Yaskawa INFORM job: sSwarf1_multiple_spiral.JBI

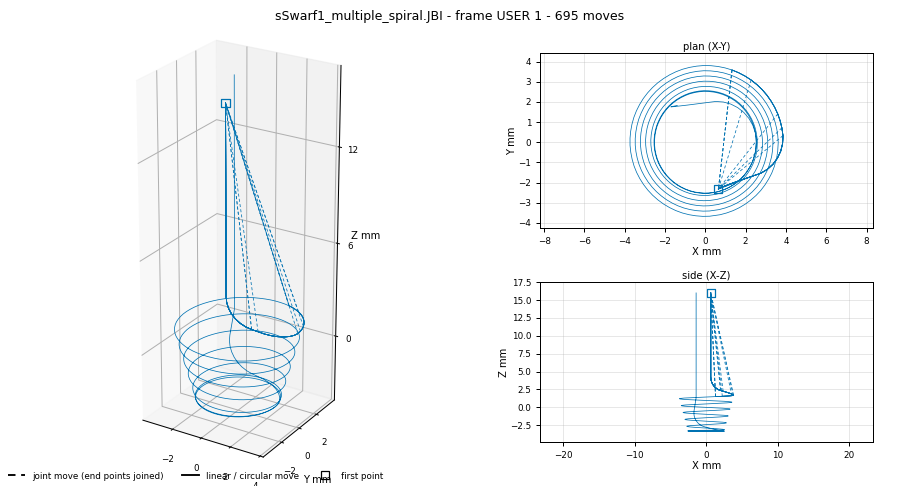
[picture p0: tool path of sSwarf1_multiple_spiral.JBI in frame USER 1, 695 of 695 moves have a stored position in this frame; points joined in program order, loops and branches not executed]
/JOB
//NAME sSwarf1_multiple_spiral
//POS
///NPOS 499,0,0,0,0,0
///USER 1
///TOOL 8
///POSTYPE USER
///RECTAN
///RCONF 1,0,0,0,0,0
C00000=50.999,-29.823,15.536,-90.000,-150.794,-116.565
C00001=50.999,-21.274,0.729,-90.000,-150.794,-116.565
C00002=50.999,-20.274,-1.003,-90.000,-150.794,-116.565
C00003=47.666,-20.274,-1.003,-90.000,-150.794,-116.565
C00004=44.332,-20.274,-1.003,-90.000,-150.794,-116.565
C00005=40.999,-20.274,-1.003,-90.000,-150.794,-116.565
C00006=36.223,-20.274,-1.003,-90.000,-150.794,-116.565
C00007=31.447,-20.274,-1.003,-90.000,-150.794,-116.565
C00008=26.671,-20.274,-1.003,-90.000,-150.794,-116.565
C00009=21.896,-20.274,-1.003,-90.000,-150.794,-116.565
C00010=17.120,-20.274,-1.003,-90.000,-150.794,-116.565
C00011=12.344,-20.274,-1.003,-90.000,-150.794,-116.565
C00012=7.568,-20.274,-1.003,-90.000,-150.794,-116.565
C00013=2.792,-20.274,-1.003,-90.000,-150.794,-116.565
C00014=-1.983,-20.274,-1.003,-90.000,-150.794,-116.565
C00015=-6.759,-20.274,-1.003,-90.000,-150.794,-116.565
C00016=-11.535,-20.274,-1.003,-90.000,-150.794,-116.565
C00017=-16.311,-20.274,-1.003,-90.000,-150.794,-116.565
C00018=-21.087,-20.274,-1.003,-90.000,-150.794,-116.565
C00019=-25.862,-20.274,-1.003,-90.000,-150.794,-116.565
C00020=-30.638,-20.274,-1.003,-90.000,-150.794,-116.565
C00021=-35.414,-20.274,-1.003,-90.000,-150.794,-116.565
C00022=-40.190,-20.274,-1.003,-90.000,-150.794,-116.565
C00023=-44.966,-20.274,-1.003,-90.000,-150.794,-116.565
C00024=-48.299,-20.274,-1.003,-90.000,-150.794,-116.565
C00025=-51.632,-20.274,-1.003,-90.000,-150.794,-116.565
C00026=-54.966,-20.274,-1.003,-90.000,-150.794,-116.565
C00027=-54.966,-21.274,0.729,-90.000,-150.794,-116.565
C00028=-54.966,-29.823,15.536,-90.000,-150.794,-116.565
C00000=53.984,-29.817,15.539,-90.000,-150.794,-116.565
C00001=53.984,-24.817,6.879,-90.000,-150.794,-116.565
C00002=53.984,-20.744,-0.175,-90.000,-150.794,-116.565
C00003=53.705,-20.407,-0.758,-90.000,-150.794,-116.565
C00004=53.031,-20.268,-1.000,-90.000,-150.794,-116.565
C00005=-55.536,-20.268,-1.000,-90.000,-150.794,-116.565
C00006=-56.209,-20.407,-0.758,-90.000,-150.794,-116.565
C00007=-56.488,-20.744,-0.175,-90.000,-150.794,-116.565
C00008=-56.488,-29.817,15.539,-90.000,-150.794,-116.565
C00000=-54.823,-30.003,15.536,180.000,-152.507,146.310
C00001=-46.274,-30.003,0.729,180.000,-152.507,146.310
C00002=-45.274,-30.003,-1.003,180.000,-152.507,146.310
C00003=-45.274,-26.669,-1.003,180.000,-152.507,146.310
C00004=-45.274,-23.336,-1.003,180.000,-152.507,146.310
C00005=-45.274,-20.003,-1.003,180.000,-152.507,146.310
C00006=-45.274,-15.558,-1.003,180.000,-152.507,146.310
C00007=-45.274,-11.113,-1.003,180.000,-152.507,146.310
C00008=-45.274,-6.668,-1.003,180.000,-152.507,146.310
C00009=-45.274,-2.223,-1.003,180.000,-152.507,146.310
C00010=-45.274,2.223,-1.003,180.000,-152.507,146.310
C00011=-45.274,6.668,-1.003,180.000,-152.507,146.310
C00012=-45.274,11.113,-1.003,180.000,-152.507,146.310
C00013=-45.274,15.558,-1.003,180.000,-152.507,146.310
C00014=-45.274,20.003,-1.003,-180.000,-152.507,146.310
C00015=-45.274,23.336,-1.003,-180.000,-152.507,146.310
C00016=-45.274,26.669,-1.003,-180.000,-152.507,146.310
C00017=-45.274,30.003,-1.003,-180.000,-152.507,146.310
C00018=-46.274,30.003,0.729,-180.000,-152.507,146.310
C00019=-54.823,30.003,15.536,-180.000,-152.507,146.310
C00000=54.301,-29.817,15.539,-90.000,-150.794,-116.565
C00001=54.301,-24.817,6.879,-90.000,-150.794,-116.565
C00002=54.301,-20.903,0.100,-90.000,-150.794,-116.565
C00003=53.929,-20.454,-0.678,-90.000,-150.794,-116.565
C00004=53.031,-20.268,-1.000,-90.000,-150.794,-116.565
C00005=-55.536,-20.268,-1.000,-90.000,-150.794,-116.565
C00006=-56.434,-20.454,-0.678,-90.000,-150.794,-116.565
C00007=-56.806,-20.903,0.100,-90.000,-150.794,-116.565
C00008=-56.806,-29.817,15.539,-90.000,-150.794,-116.565
C00000=-54.969,29.823,15.536,90.000,-150.794,63.435
C00001=-54.969,21.274,0.729,90.000,-150.794,63.435
C00002=-54.969,20.274,-1.003,90.000,-150.794,63.435
C00003=-51.636,20.274,-1.003,90.000,-150.794,63.435
C00004=-48.303,20.274,-1.003,90.000,-150.794,63.435
C00005=-44.969,20.274,-1.003,90.000,-150.794,63.435
C00006=-40.029,20.274,-1.003,90.000,-150.794,63.435
C00007=-35.088,20.274,-1.003,90.000,-150.794,63.435
C00008=-30.147,20.274,-1.003,90.000,-150.794,63.435
C00009=-25.206,20.274,-1.003,90.000,-150.794,63.435
C00010=-20.266,20.274,-1.003,90.000,-150.794,63.435
C00011=-15.325,20.274,-1.003,90.000,-150.794,63.435
C00012=-10.384,20.274,-1.003,90.000,-150.794,63.435
C00013=-5.443,20.274,-1.003,90.000,-150.794,63.435
C00014=-0.502,20.274,-1.003,90.000,-150.794,63.435
C00015=4.438,20.274,-1.003,90.000,-150.794,63.435
C00016=9.379,20.274,-1.003,90.000,-150.794,63.435
C00017=14.320,20.274,-1.003,90.000,-150.794,63.435
C00018=19.261,20.274,-1.003,90.000,-150.794,63.435
C00019=24.201,20.274,-1.003,90.000,-150.794,63.435
C00020=29.142,20.274,-1.003,90.000,-150.794,63.435
C00021=34.083,20.274,-1.003,90.000,-150.794,63.435
C00022=39.024,20.274,-1.003,90.000,-150.794,63.435
C00023=43.965,20.274,-1.003,90.000,-150.794,63.435
C00024=47.298,20.274,-1.003,90.000,-150.794,63.435
C00025=50.631,20.274,-1.003,90.000,-150.794,63.435
C00026=53.965,20.274,-1.003,90.000,-150.794,63.435
C00027=53.965,21.274,0.729,90.000,-150.794,63.435
C00028=53.965,29.823,15.536,90.000,-150.794,63.435
C00000=-54.969,29.823,15.536,90.000,-150.794,63.435
C00001=-54.969,21.274,0.729,90.000,-150.794,63.435
C00002=-54.969,20.274,-1.003,90.000,-150.794,63.435
C00003=-51.636,20.274,-1.003,90.000,-150.794,63.435
C00004=-48.303,20.274,-1.003,90.000,-150.794,63.435
C00005=-44.969,20.274,-1.003,90.000,-150.794,63.435
C00006=-40.029,20.274,-1.003,90.000,-150.794,63.435
C00007=-35.088,20.274,-1.003,90.000,-150.794,63.435
C00008=-30.147,20.274,-1.003,90.000,-150.794,63.435
C00009=-25.206,20.274,-1.003,90.000,-150.794,63.435
C00010=-20.266,20.274,-1.003,90.000,-150.794,63.435
C00011=-15.325,20.274,-1.003,90.000,-150.794,63.435
C00012=-10.384,20.274,-1.003,90.000,-150.794,63.435
C00013=-5.443,20.274,-1.003,90.000,-150.794,63.435
C00014=-0.502,20.274,-1.003,90.000,-150.794,63.435
C00015=4.438,20.274,-1.003,90.000,-150.794,63.435
C00016=9.379,20.274,-1.003,90.000,-150.794,63.435
C00017=14.320,20.274,-1.003,90.000,-150.794,63.435
C00018=19.261,20.274,-1.003,90.000,-150.794,63.435
C00019=24.201,20.274,-1.003,90.000,-150.794,63.435
C00020=29.142,20.274,-1.003,90.000,-150.794,63.435
C00021=34.083,20.274,-1.003,90.000,-150.794,63.435
C00022=39.024,20.274,-1.003,90.000,-150.794,63.435
C00023=43.965,20.274,-1.003,90.000,-150.794,63.435
C00024=47.298,20.274,-1.003,90.000,-150.794,63.435
C00025=50.631,20.274,-1.003,90.000,-150.794,63.435
C00026=53.965,20.274,-1.003,90.000,-150.794,63.435
C00027=53.965,21.274,0.729,90.000,-150.794,63.435
C00028=53.965,29.823,15.536,90.000,-150.794,63.435
C00000=54.817,28.503,15.539,0.000,-152.507,-33.690
C00001=46.268,28.503,0.732,0.000,-152.507,-33.690
C00002=45.268,28.503,-1.000,0.000,-152.507,-33.690
C00003=45.268,25.169,-1.000,0.000,-152.507,-33.690
C00004=45.268,21.836,-1.000,0.000,-152.507,-33.690
C00005=45.268,18.503,-1.000,0.000,-152.507,-33.690
C00006=45.268,13.573,-1.000,0.000,-152.507,-33.690
C00007=45.268,8.644,-1.000,0.000,-152.507,-33.690
C00008=45.268,3.715,-1.000,0.000,-152.507,-33.690
C00009=45.268,-1.214,-1.000,0.000,-152.507,-33.690
C00010=45.268,-6.144,-1.000,0.000,-152.507,-33.690
C00011=45.268,-11.073,-1.000,0.000,-152.507,-33.690
C00012=45.268,-16.002,-1.000,0.000,-152.507,-33.690
C00013=45.268,-19.336,-1.000,0.000,-152.507,-33.690
C00014=45.268,-22.669,-1.000,0.000,-152.507,-33.690
C00015=45.268,-26.002,-1.000,0.000,-152.507,-33.690
C00016=46.268,-26.002,0.732,0.000,-152.507,-33.690
C00017=54.817,-26.002,15.539,0.000,-152.507,-33.690
C00000=54.817,28.728,15.539,0.000,-152.507,-33.690
C00001=46.268,28.728,0.732,0.000,-152.507,-33.690
C00002=45.268,28.728,-1.000,0.000,-152.507,-33.690
C00003=45.268,25.395,-1.000,0.000,-152.507,-33.690
C00004=45.268,22.062,-1.000,0.000,-152.507,-33.690
C00005=45.268,18.728,-1.000,0.000,-152.507,-33.690
C00006=45.268,13.751,-1.000,0.000,-152.507,-33.690
C00007=45.268,8.773,-1.000,0.000,-152.507,-33.690
C00008=45.268,3.795,-1.000,0.000,-152.507,-33.690
C00009=45.268,-1.182,-1.000,0.000,-152.507,-33.690
C00010=45.268,-6.160,-1.000,0.000,-152.507,-33.690
C00011=45.268,-11.138,-1.000,0.000,-152.507,-33.690
C00012=45.268,-16.115,-1.000,0.000,-152.507,-33.690
C00013=45.268,-21.115,-1.000,0.000,-152.507,-33.690
C00014=45.268,-26.115,-1.000,0.000,-152.507,-33.690
C00015=46.268,-26.115,0.732,0.000,-152.507,-33.690
C00016=54.817,-26.115,15.539,0.000,-152.507,-33.690
C00000=43.731,-18.731,20.821,-45.000,-157.889,-76.068
C00001=38.802,-13.802,3.748,-45.000,-157.889,-76.068
C00002=38.268,-13.268,1.896,-45.000,-157.889,-76.068
C00003=41.541,-16.541,0.006,-45.000,-157.889,-76.068
C00004=44.127,-19.127,-1.487,-45.000,-157.889,-76.068
C00005=46.712,-21.712,-2.979,-44.999,-157.889,-76.067
C00006=49.985,-24.985,-4.869,-44.999,-157.889,-76.067
C00007=50.520,-25.520,-3.018,-44.999,-157.889,-76.067
C00008=50.520,-25.520,-3.018,-44.999,-157.889,-76.067
C00009=55.449,-30.449,14.056,-44.999,-157.889,-76.067
C00000=-1.500,-1.270,16.240,0.000,-180.000,-30.000
C00001=-1.500,-1.270,6.080,0.000,-180.000,-30.000
C00002=-1.500,-1.270,2.000,0.000,-180.000,-30.000
C00003=-1.500,-1.270,-3.730,0.000,-180.000,-30.000
C00004=-1.128,-1.270,-4.628,0.000,-180.000,-30.000
C00005=-0.230,-1.270,-5.000,0.000,-180.000,-30.000
C00006=1.040,-1.270,-5.000,0.000,-180.000,-30.000
C00007=1.938,-0.898,-5.000,0.000,-180.000,-30.000
C00008=2.310,0.000,-5.000,0.000,-180.000,-30.000
C00009=1.944,1.249,-5.000,0.000,-180.000,-30.000
C00010=0.960,2.101,-5.000,0.000,-180.000,-30.000
C00011=-0.329,2.287,-5.000,0.000,-180.000,-30.000
C00012=-1.513,1.746,-5.000,0.000,-180.000,-30.000
C00013=-2.217,0.651,-5.000,0.000,-180.000,-30.000
C00014=-2.217,-0.651,-5.000,0.000,-180.000,-30.000
C00015=-1.513,-1.746,-5.000,0.000,-180.000,-30.000
C00016=-0.329,-2.287,-5.000,0.000,-180.000,-30.000
C00017=0.960,-2.101,-5.000,0.000,-180.000,-30.000
C00018=1.944,-1.249,-5.000,0.000,-180.000,-30.000
C00019=2.310,0.000,-5.000,0.000,-180.000,-30.000
C00020=1.938,0.898,-5.000,0.000,-180.000,-30.000
C00021=1.040,1.270,-5.000,0.000,-180.000,-30.000
C00022=-0.230,1.270,-5.000,0.000,-180.000,-30.000
C00023=-1.128,1.270,-4.628,0.000,-180.000,-30.000
C00024=-1.500,1.270,-3.730,0.000,-180.000,-30.000
C00025=-1.500,1.270,16.240,0.000,-180.000,-30.000
C00000=0.647,-2.321,16.000,5.978,-170.659,-24.314
C00001=0.647,-2.321,4.269,5.978,-170.659,-24.314
C00002=0.675,-2.297,3.898,5.978,-170.659,-24.314
C00003=0.769,-2.252,3.540,5.978,-170.659,-24.314
C00004=0.924,-2.188,3.208,5.978,-170.659,-24.314
C00005=1.136,-2.106,2.912,5.978,-170.659,-24.314
C00006=1.396,-2.010,2.663,5.978,-170.659,-24.314
C00007=1.697,-1.902,2.470,5.978,-170.659,-24.314
C00008=2.027,-1.787,2.340,5.978,-170.659,-24.314
C00009=2.385,-1.664,2.237,6.753,-170.076,-23.570
C00010=2.743,-1.541,2.135,7.489,-169.489,-22.867
C00011=3.069,-1.349,2.034,4.077,-168.639,-26.386
C00012=3.351,-1.094,1.937,2.800,-167.769,-27.759
C00013=3.578,-0.786,1.849,2.935,-166.964,-27.702
C00014=3.740,-0.438,1.773,4.077,-166.295,-26.612
C00015=3.833,-0.062,1.712,5.891,-165.805,-24.815
C00016=3.851,0.328,1.668,8.109,-165.519,-22.577
C00017=3.795,0.715,1.643,10.503,-165.449,-20.129
C00018=3.710,1.065,1.629,15.772,-165.465,-14.708
C00019=3.591,1.406,1.616,21.045,-165.470,-9.266
C00020=3.440,1.733,1.601,26.330,-165.496,-3.799
C00021=3.259,2.044,1.586,31.634,-165.496,1.692
C00022=3.052,2.338,1.571,36.954,-165.487,7.196
C00023=2.818,2.610,1.558,42.300,-165.472,12.720
C00024=2.559,2.858,1.543,47.675,-165.442,18.258
C00025=2.270,3.089,1.527,53.385,-165.428,24.116
C00026=1.968,3.283,1.513,58.665,-165.382,29.508
C00027=1.652,3.449,1.500,63.941,-165.340,34.866
C00028=1.322,3.586,1.485,69.220,-165.289,40.196
C00029=0.980,3.689,1.471,74.498,-165.249,45.490
C00030=0.630,3.759,1.456,79.782,-165.218,50.757
C00031=0.276,3.799,1.442,85.071,-165.158,55.997
C00032=-0.079,3.807,1.428,90.352,-165.106,61.200
C00033=-0.434,3.776,1.413,95.641,-165.093,66.377
C00034=-0.784,3.715,1.398,100.933,-165.058,71.538
C00035=-1.127,3.624,1.384,106.227,-165.039,76.679
C00036=-1.458,3.499,1.371,111.524,-165.001,81.809
C00037=-1.776,3.343,1.356,116.817,-165.007,86.925
C00038=-2.079,3.159,1.341,122.121,-165.009,92.049
C00039=-2.363,2.949,1.327,127.425,-165.005,97.175
C00040=-2.625,2.713,1.313,132.730,-165.023,102.310
C00041=-2.864,2.453,1.299,138.038,-165.041,107.460
C00042=-3.078,2.173,1.283,143.347,-165.074,112.632
C00043=-3.263,1.873,1.269,148.665,-165.122,117.838
C00044=-3.421,1.559,1.256,153.984,-165.142,123.069
C00045=-3.549,1.232,1.241,159.299,-165.195,128.330
C00046=-3.643,0.894,1.226,164.626,-165.238,133.634
C00047=-3.706,0.549,1.212,169.954,-165.291,138.974
C00048=-3.739,0.201,1.198,175.289,-165.326,144.353
C00049=-3.739,-0.149,1.184,-179.378,-165.350,149.762
C00050=-3.702,-0.497,1.169,-174.043,-165.412,155.210
C00051=-3.635,-0.840,1.154,-168.695,-165.440,160.694
C00052=-3.540,-1.175,1.140,-163.348,-165.455,166.199
C00053=-3.411,-1.499,1.126,-157.996,-165.474,171.725
C00054=-3.251,-1.808,1.111,-152.641,-165.485,177.266
C00055=-3.065,-2.102,1.096,-147.279,-165.500,-177.183
C00056=-2.853,-2.377,1.082,-141.904,-165.474,-171.622
C00057=-2.616,-2.630,1.069,-136.533,-165.456,-166.075
C00058=-2.357,-2.859,1.054,-131.152,-165.437,-160.536
C00059=-2.078,-3.064,1.039,-125.763,-165.399,-155.010
C00060=-1.780,-3.240,1.025,-120.366,-165.375,-149.505
C00061=-1.469,-3.390,1.011,-114.956,-165.317,-144.016
C00062=-1.145,-3.509,0.997,-109.545,-165.274,-138.561
C00063=-0.812,-3.595,0.981,-104.115,-165.244,-133.124
C00064=-0.472,-3.650,0.967,-98.666,-165.194,-127.701
C00065=-0.129,-3.677,0.953,-93.198,-165.150,-122.295
C00066=0.214,-3.670,0.939,-87.702,-165.092,-116.891
C00067=0.727,-3.597,0.916,-79.195,-165.071,-108.588
C00068=1.058,-3.508,0.903,-73.856,-165.034,-103.402
C00069=1.380,-3.392,0.889,-68.517,-165.012,-98.231
C00070=1.689,-3.245,0.874,-63.171,-165.000,-93.064
C00071=1.981,-3.069,0.859,-57.818,-165.006,-87.892
C00072=2.256,-2.867,0.845,-52.451,-165.024,-82.705
C00073=2.513,-2.642,0.832,-47.075,-165.019,-77.501
C00074=2.746,-2.395,0.817,-41.695,-165.044,-72.279
C00075=2.952,-2.124,0.802,-36.294,-165.092,-67.015
C00076=3.134,-1.837,0.787,-30.877,-165.124,-61.712
C00077=3.291,-1.536,0.773,-25.437,-165.164,-56.358
C00078=3.415,-1.221,0.760,-19.970,-165.193,-50.946
C00079=3.539,-0.772,0.738,-12.233,-165.284,-43.221
C00080=3.590,-0.437,0.724,-6.959,-165.319,-37.916
C00081=3.615,-0.003,0.707,0.000,-165.365,-30.867
C00082=3.592,0.334,0.692,5.247,-165.405,-25.517
C00083=3.541,0.668,0.677,10.503,-165.449,-20.129
C00084=3.461,0.995,0.663,15.772,-165.465,-14.708
C00085=3.350,1.313,0.650,21.045,-165.470,-9.266
C00086=3.208,1.618,0.635,26.330,-165.496,-3.799
C00087=3.039,1.908,0.620,31.634,-165.496,1.692
C00088=2.846,2.182,0.605,36.954,-165.487,7.196
C00089=2.626,2.436,0.592,42.300,-165.472,12.720
C00090=2.385,2.667,0.577,47.675,-165.442,18.258
C00091=2.116,2.882,0.561,53.385,-165.428,24.116
C00092=1.834,3.062,0.547,58.665,-165.382,29.508
C00093=1.538,3.217,0.534,63.941,-165.340,34.866
C00094=1.230,3.344,0.519,69.220,-165.289,40.196
C00095=0.911,3.440,0.505,74.498,-165.249,45.490
C00096=0.585,3.505,0.490,79.782,-165.218,50.757
C00097=0.254,3.541,0.476,85.071,-165.158,55.997
C00098=-0.078,3.548,0.462,90.352,-165.106,61.200
C00099=-0.408,3.519,0.447,95.641,-165.093,66.377
C00100=-0.734,3.461,0.432,100.933,-165.058,71.538
C00101=-1.054,3.375,0.418,106.227,-165.039,76.679
C00102=-1.363,3.258,0.405,111.524,-165.001,81.809
C00103=-1.660,3.112,0.390,116.817,-165.007,86.925
C00104=-1.941,2.940,0.374,122.121,-165.009,92.049
C00105=-2.205,2.743,0.361,127.425,-165.005,97.175
C00106=-2.449,2.522,0.347,132.730,-165.023,102.310
C00107=-2.671,2.280,0.332,138.038,-165.041,107.460
C00108=-2.870,2.019,0.317,143.347,-165.074,112.632
C00109=-3.042,1.739,0.303,148.665,-165.122,117.838
C00110=-3.188,1.446,0.289,153.984,-165.142,123.069
C00111=-3.307,1.141,0.275,159.299,-165.195,128.330
C00112=-3.393,0.825,0.260,164.626,-165.238,133.634
C00113=-3.451,0.504,0.245,169.954,-165.291,138.974
C00114=-3.481,0.179,0.232,175.289,-165.326,144.353
C00115=-3.480,-0.146,0.218,-179.378,-165.350,149.762
C00116=-3.445,-0.470,0.202,-174.043,-165.412,155.210
C00117=-3.382,-0.789,0.188,-168.695,-165.440,160.694
C00118=-3.291,-1.101,0.174,-163.348,-165.455,166.199
C00119=-3.171,-1.402,0.160,-157.996,-165.474,171.725
C00120=-3.021,-1.689,0.145,-152.641,-165.485,177.266
C00121=-2.848,-1.962,0.130,-147.279,-165.500,-177.183
C00122=-2.649,-2.217,0.116,-141.904,-165.474,-171.622
C00123=-2.428,-2.452,0.103,-136.533,-165.456,-166.075
C00124=-2.186,-2.664,0.088,-131.152,-165.437,-160.536
C00125=-1.926,-2.854,0.073,-125.763,-165.399,-155.010
C00126=-1.649,-3.017,0.059,-120.366,-165.375,-149.505
C00127=-1.359,-3.155,0.045,-114.956,-165.317,-144.016
C00128=-1.058,-3.265,0.031,-109.545,-165.274,-138.561
C00129=-0.748,-3.344,0.015,-104.115,-165.244,-133.124
C00130=-0.433,-3.395,0.001,-98.666,-165.194,-127.701
C00131=-0.115,-3.418,-0.013,-93.198,-165.150,-122.295
C00132=0.203,-3.411,-0.027,-87.702,-165.092,-116.891
C00133=0.678,-3.343,-0.050,-79.195,-165.071,-108.588
C00134=0.986,-3.260,-0.063,-73.856,-165.034,-103.402
C00135=1.285,-3.151,-0.077,-68.517,-165.012,-98.231
C00136=1.572,-3.014,-0.092,-63.171,-165.000,-93.064
C00137=1.844,-2.850,-0.107,-57.818,-165.006,-87.892
C00138=2.099,-2.662,-0.121,-52.451,-165.024,-82.705
C00139=2.336,-2.453,-0.134,-47.075,-165.019,-77.501
C00140=2.553,-2.222,-0.149,-41.695,-165.044,-72.279
C00141=2.744,-1.971,-0.164,-36.294,-165.092,-67.015
C00142=2.912,-1.704,-0.179,-30.877,-165.124,-61.712
C00143=3.057,-1.425,-0.193,-25.437,-165.164,-56.358
C00144=3.172,-1.133,-0.206,-19.970,-165.193,-50.946
C00145=3.286,-0.717,-0.228,-12.233,-165.284,-43.221
C00146=3.333,-0.406,-0.242,-6.959,-165.319,-37.916
C00147=3.357,-0.003,-0.259,0.000,-165.365,-30.867
C00148=3.335,0.310,-0.274,5.247,-165.405,-25.517
C00149=3.287,0.621,-0.289,10.503,-165.449,-20.129
C00150=3.212,0.925,-0.303,15.772,-165.465,-14.708
C00151=3.108,1.220,-0.316,21.045,-165.470,-9.266
C00152=2.976,1.503,-0.332,26.330,-165.496,-3.799
C00153=2.819,1.773,-0.346,31.634,-165.496,1.692
C00154=2.639,2.027,-0.361,36.954,-165.487,7.196
C00155=2.435,2.261,-0.374,42.300,-165.472,12.720
C00156=2.210,2.475,-0.389,47.675,-165.442,18.258
C00157=1.961,2.674,-0.405,53.385,-165.428,24.116
C00158=1.699,2.841,-0.419,58.665,-165.382,29.508
C00159=1.425,2.984,-0.432,63.941,-165.340,34.866
C00160=1.138,3.102,-0.447,69.220,-165.289,40.196
C00161=0.842,3.190,-0.462,74.498,-165.249,45.490
C00162=0.539,3.250,-0.477,79.782,-165.218,50.757
C00163=0.232,3.283,-0.490,85.071,-165.158,55.997
C00164=-0.076,3.289,-0.504,90.352,-165.106,61.200
C00165=-0.383,3.261,-0.519,95.641,-165.093,66.377
C00166=-0.685,3.206,-0.534,100.933,-165.058,71.538
C00167=-0.982,3.127,-0.548,106.227,-165.039,76.679
C00168=-1.268,3.017,-0.562,111.524,-165.001,81.809
C00169=-1.543,2.881,-0.577,116.817,-165.007,86.925
C00170=-1.804,2.721,-0.592,122.121,-165.009,92.049
C00171=-2.048,2.538,-0.605,127.425,-165.005,97.175
C00172=-2.274,2.332,-0.619,132.730,-165.023,102.310
C00173=-2.479,2.107,-0.634,138.038,-165.041,107.460
C00174=-2.663,1.864,-0.649,143.347,-165.074,112.632
C00175=-2.821,1.604,-0.664,148.665,-165.122,117.838
C00176=-2.955,1.332,-0.677,153.984,-165.142,123.069
C00177=-3.065,1.049,-0.692,159.299,-165.195,128.330
C00178=-3.144,0.757,-0.707,164.626,-165.238,133.634
C00179=-3.196,0.459,-0.721,169.954,-165.291,138.974
C00180=-3.223,0.158,-0.735,175.289,-165.326,144.353
C00181=-3.220,-0.144,-0.748,-179.378,-165.350,149.762
C00182=-3.187,-0.443,-0.764,-174.043,-165.412,155.210
C00183=-3.128,-0.738,-0.778,-168.695,-165.440,160.694
C00184=-3.043,-1.026,-0.792,-163.348,-165.455,166.199
C00185=-2.931,-1.305,-0.806,-157.996,-165.474,171.725
C00186=-2.791,-1.570,-0.821,-152.641,-165.485,177.266
C00187=-2.630,-1.822,-0.837,-147.279,-165.500,-177.183
C00188=-2.446,-2.057,-0.850,-141.904,-165.474,-171.622
C00189=-2.240,-2.273,-0.864,-136.533,-165.456,-166.075
C00190=-2.016,-2.469,-0.879,-131.152,-165.437,-160.536
C00191=-1.775,-2.644,-0.893,-125.763,-165.399,-155.010
C00192=-1.518,-2.794,-0.908,-120.366,-165.375,-149.505
C00193=-1.250,-2.920,-0.921,-114.956,-165.317,-144.016
C00194=-0.972,-3.021,-0.936,-109.545,-165.274,-138.561
C00195=-0.685,-3.093,-0.951,-104.115,-165.244,-133.124
C00196=-0.394,-3.139,-0.965,-98.666,-165.194,-127.701
C00197=-0.100,-3.160,-0.979,-93.198,-165.150,-122.295
C00198=0.193,-3.152,-0.993,-87.702,-165.092,-116.891
C00199=0.630,-3.089,-1.016,-79.195,-165.071,-108.588
C00200=0.914,-3.011,-1.030,-73.856,-165.034,-103.402
C00201=1.190,-2.910,-1.043,-68.517,-165.012,-98.231
C00202=1.455,-2.783,-1.058,-63.171,-165.000,-93.064
C00203=1.706,-2.631,-1.073,-57.818,-165.006,-87.892
C00204=1.941,-2.457,-1.087,-52.451,-165.024,-82.705
C00205=2.160,-2.263,-1.100,-47.075,-165.019,-77.501
C00206=2.360,-2.050,-1.115,-41.695,-165.044,-72.279
C00207=2.535,-1.818,-1.130,-36.294,-165.092,-67.015
C00208=2.690,-1.572,-1.145,-30.877,-165.124,-61.712
C00209=2.823,-1.314,-1.159,-25.437,-165.164,-56.358
C00210=2.929,-1.045,-1.172,-19.970,-165.193,-50.946
C00211=3.034,-0.662,-1.194,-12.233,-165.284,-43.221
C00212=3.076,-0.374,-1.207,-6.959,-165.319,-37.916
C00213=3.098,-0.003,-1.225,0.000,-165.365,-30.867
C00214=3.077,0.287,-1.240,5.247,-165.405,-25.517
C00215=3.033,0.573,-1.255,10.503,-165.449,-20.129
C00216=2.963,0.854,-1.269,15.772,-165.465,-14.708
C00217=2.866,1.127,-1.282,21.045,-165.470,-9.266
C00218=2.744,1.388,-1.298,26.330,-165.496,-3.799
C00219=2.599,1.637,-1.312,31.634,-165.496,1.692
C00220=2.432,1.871,-1.327,36.954,-165.487,7.196
C00221=2.243,2.087,-1.340,42.300,-165.472,12.720
C00222=2.036,2.284,-1.355,47.675,-165.442,18.258
C00223=1.807,2.467,-1.371,53.385,-165.428,24.116
C00224=1.565,2.620,-1.385,58.665,-165.382,29.508
C00225=1.311,2.752,-1.398,63.941,-165.340,34.866
C00226=1.047,2.860,-1.413,69.220,-165.289,40.196
C00227=0.773,2.941,-1.428,74.498,-165.249,45.490
C00228=0.493,2.996,-1.443,79.782,-165.218,50.757
C00229=0.210,3.026,-1.456,85.071,-165.158,55.997
C00230=-0.075,3.030,-1.470,90.352,-165.106,61.200
C00231=-0.357,3.004,-1.486,95.641,-165.093,66.377
C00232=-0.636,2.952,-1.500,100.933,-165.058,71.538
C00233=-0.910,2.879,-1.515,106.227,-165.039,76.679
C00234=-1.173,2.776,-1.528,111.524,-165.001,81.809
C00235=-1.426,2.650,-1.543,116.817,-165.007,86.925
C00236=-1.666,2.502,-1.558,122.121,-165.009,92.049
C00237=-1.891,2.332,-1.572,127.425,-165.005,97.175
C00238=-2.098,2.142,-1.586,132.730,-165.023,102.310
C00239=-2.286,1.934,-1.600,138.038,-165.041,107.460
C00240=-2.455,1.709,-1.615,143.347,-165.074,112.632
C00241=-2.600,1.470,-1.630,148.665,-165.122,117.838
C00242=-2.722,1.218,-1.643,153.984,-165.142,123.069
C00243=-2.822,0.958,-1.658,159.299,-165.195,128.330
C00244=-2.894,0.688,-1.673,164.626,-165.238,133.634
C00245=-2.941,0.414,-1.687,169.954,-165.291,138.974
C00246=-2.965,0.137,-1.701,175.289,-165.326,144.353
C00247=-2.961,-0.141,-1.714,-179.378,-165.350,149.762
C00248=-2.930,-0.416,-1.730,-174.043,-165.412,155.210
C00249=-2.874,-0.687,-1.745,-168.695,-165.440,160.694
C00250=-2.795,-0.952,-1.758,-163.348,-165.455,166.199
C00251=-2.690,-1.207,-1.773,-157.996,-165.474,171.725
C00252=-2.561,-1.451,-1.787,-152.641,-165.485,177.266
C00253=-2.412,-1.682,-1.803,-147.279,-165.500,-177.183
C00254=-2.242,-1.897,-1.816,-141.904,-165.474,-171.622
C00255=-2.052,-2.095,-1.830,-136.533,-165.456,-166.075
C00256=-1.846,-2.275,-1.845,-131.152,-165.437,-160.536
C00257=-1.624,-2.434,-1.859,-125.763,-165.399,-155.010
C00258=-1.388,-2.570,-1.874,-120.366,-165.375,-149.505
C00259=-1.141,-2.685,-1.887,-114.956,-165.317,-144.016
C00260=-0.885,-2.777,-1.902,-109.545,-165.274,-138.561
C00261=-0.622,-2.843,-1.917,-104.115,-165.244,-133.124
C00262=-0.355,-2.883,-1.931,-98.666,-165.194,-127.701
C00263=-0.086,-2.901,-1.945,-93.198,-165.150,-122.295
C00264=0.183,-2.893,-1.959,-87.702,-165.092,-116.891
C00265=0.581,-2.835,-1.982,-79.195,-165.071,-108.588
C00266=0.842,-2.763,-1.996,-73.856,-165.034,-103.402
C00267=1.095,-2.669,-2.009,-68.517,-165.012,-98.231
C00268=1.338,-2.552,-2.024,-63.171,-165.000,-93.064
C00269=1.568,-2.412,-2.039,-57.818,-165.006,-87.892
C00270=1.784,-2.252,-2.053,-52.451,-165.024,-82.705
C00271=1.984,-2.073,-2.067,-47.075,-165.019,-77.501
C00272=2.166,-1.878,-2.081,-41.695,-165.044,-72.279
C00273=2.327,-1.665,-2.097,-36.294,-165.092,-67.015
C00274=2.468,-1.439,-2.111,-30.877,-165.124,-61.712
C00275=2.590,-1.203,-2.125,-25.437,-165.164,-56.358
C00276=2.685,-0.956,-2.138,-19.970,-165.193,-50.946
C00277=2.781,-0.608,-2.160,-12.233,-165.284,-43.221
C00278=2.819,-0.343,-2.173,-6.959,-165.319,-37.916
C00279=2.839,-0.003,-2.191,0.000,-165.365,-30.867
C00280=2.819,0.263,-2.206,5.247,-165.405,-25.517
C00281=2.778,0.526,-2.221,10.503,-165.449,-20.129
C00282=2.714,0.784,-2.235,15.772,-165.465,-14.708
C00283=2.625,1.034,-2.248,21.045,-165.470,-9.266
C00284=2.512,1.274,-2.264,26.330,-165.496,-3.799
C00285=2.378,1.501,-2.278,31.634,-165.496,1.692
C00286=2.225,1.716,-2.293,36.954,-165.487,7.196
C00287=2.052,1.913,-2.306,42.300,-165.472,12.720
C00288=1.862,2.093,-2.321,47.675,-165.442,18.258
C00289=1.653,2.259,-2.337,53.385,-165.428,24.116
C00290=1.430,2.399,-2.351,58.665,-165.382,29.508
C00291=1.197,2.519,-2.364,63.941,-165.340,34.866
C00292=0.955,2.618,-2.379,69.220,-165.289,40.196
C00293=0.703,2.691,-2.394,74.498,-165.249,45.490
C00294=0.447,2.741,-2.409,79.782,-165.218,50.757
C00295=0.187,2.768,-2.422,85.071,-165.158,55.997
C00296=-0.073,2.771,-2.436,90.352,-165.106,61.200
C00297=-0.332,2.746,-2.452,95.641,-165.093,66.377
C00298=-0.587,2.698,-2.466,100.933,-165.058,71.538
C00299=-0.837,2.630,-2.481,106.227,-165.039,76.679
C00300=-1.078,2.535,-2.494,111.524,-165.001,81.809
C00301=-1.309,2.419,-2.509,116.817,-165.007,86.925
C00302=-1.529,2.283,-2.524,122.121,-165.009,92.049
C00303=-1.733,2.126,-2.538,127.425,-165.005,97.175
C00304=-1.922,1.952,-2.552,132.730,-165.023,102.310
C00305=-2.094,1.760,-2.566,138.038,-165.041,107.460
C00306=-2.247,1.555,-2.582,143.347,-165.074,112.632
C00307=-2.379,1.335,-2.596,148.665,-165.122,117.838
C00308=-2.489,1.105,-2.609,153.984,-165.142,123.069
C00309=-2.580,0.866,-2.624,159.299,-165.195,128.330
C00310=-2.644,0.619,-2.639,164.626,-165.238,133.634
C00311=-2.687,0.369,-2.654,169.954,-165.291,138.974
C00312=-2.707,0.115,-2.667,175.289,-165.326,144.353
C00313=-2.702,-0.138,-2.681,-179.378,-165.350,149.762
C00314=-2.672,-0.389,-2.697,-174.043,-165.412,155.210
C00315=-2.620,-0.637,-2.711,-168.695,-165.440,160.694
C00316=-2.547,-0.878,-2.725,-163.348,-165.455,166.199
C00317=-2.450,-1.110,-2.739,-157.996,-165.474,171.725
C00318=-2.331,-1.332,-2.754,-152.641,-165.485,177.266
C00319=-2.195,-1.542,-2.769,-147.279,-165.500,-177.183
C00320=-2.038,-1.737,-2.783,-141.904,-165.474,-171.622
C00321=-1.864,-1.917,-2.796,-136.533,-165.456,-166.075
C00322=-1.675,-2.080,-2.811,-131.152,-165.437,-160.536
C00323=-1.472,-2.224,-2.826,-125.763,-165.399,-155.010
C00324=-1.257,-2.347,-2.840,-120.366,-165.375,-149.505
C00325=-1.031,-2.450,-2.853,-114.956,-165.317,-144.016
C00326=-0.798,-2.533,-2.868,-109.545,-165.274,-138.561
C00327=-0.559,-2.592,-2.884,-104.115,-165.244,-133.124
C00328=-0.316,-2.627,-2.898,-98.666,-165.194,-127.701
C00329=-0.071,-2.643,-2.911,-93.198,-165.150,-122.295
C00330=0.172,-2.634,-2.925,-87.702,-165.092,-116.891
C00331=0.533,-2.581,-2.948,-79.195,-165.071,-108.588
C00332=0.770,-2.514,-2.962,-73.856,-165.034,-103.402
C00333=1.000,-2.428,-2.975,-68.517,-165.012,-98.231
C00334=1.221,-2.321,-2.990,-63.171,-165.000,-93.064
C00335=1.430,-2.193,-3.005,-57.818,-165.006,-87.892
C00336=1.626,-2.047,-3.020,-52.451,-165.024,-82.705
C00337=1.807,-1.884,-3.033,-47.075,-165.019,-77.501
C00338=1.973,-1.706,-3.047,-41.695,-165.044,-72.279
C00339=2.119,-1.512,-3.063,-36.294,-165.092,-67.015
C00340=2.246,-1.306,-3.077,-30.877,-165.124,-61.712
C00341=2.356,-1.092,-3.091,-25.437,-165.164,-56.358
C00342=2.442,-0.868,-3.104,-19.970,-165.193,-50.946
C00343=2.529,-0.553,-3.126,-12.233,-165.284,-43.221
C00344=2.563,-0.312,-3.139,-6.959,-165.319,-37.916
C00345=2.580,-0.003,-3.157,0.000,-165.365,-30.867
C00346=2.562,0.239,-3.172,5.247,-165.405,-25.517
C00347=2.524,0.479,-3.187,10.503,-165.449,-20.129
C00348=2.468,0.715,-3.189,15.772,-165.465,-14.708
C00349=2.389,0.943,-3.190,21.045,-165.470,-9.266
C00350=2.289,1.163,-3.194,26.330,-165.496,-3.799
C00351=2.169,1.372,-3.197,31.634,-165.496,1.692
C00352=2.031,1.570,-3.199,36.954,-165.487,7.196
C00353=1.875,1.752,-3.201,42.300,-165.472,12.720
C00354=1.702,1.918,-3.203,47.675,-165.442,18.258
C00355=1.514,2.072,-3.208,53.385,-165.428,24.116
C00356=1.311,2.202,-3.210,58.665,-165.382,29.508
C00357=1.098,2.316,-3.211,63.941,-165.340,34.866
C00358=0.875,2.409,-3.214,69.220,-165.289,40.196
C00359=0.645,2.479,-3.217,74.498,-165.249,45.490
C00360=0.408,2.528,-3.220,79.782,-165.218,50.757
C00361=0.169,2.554,-3.221,85.071,-165.158,55.997
C00362=-0.072,2.560,-3.223,90.352,-165.106,61.200
C00363=-0.312,2.540,-3.227,95.641,-165.093,66.377
C00364=-0.548,2.498,-3.230,100.933,-165.058,71.538
C00365=-0.781,2.437,-3.232,106.227,-165.039,76.679
C00366=-1.005,2.351,-3.234,111.524,-165.001,81.809
C00367=-1.221,2.245,-3.237,116.817,-165.007,86.925
C00368=-1.427,2.121,-3.240,122.121,-165.009,92.049
C00369=-1.619,1.977,-3.242,127.425,-165.005,97.175
C00370=-1.797,1.816,-3.244,132.730,-165.023,102.310
C00371=-1.958,1.639,-3.247,138.038,-165.041,107.460
C00372=-2.103,1.448,-3.250,143.347,-165.074,112.632
C00373=-2.229,1.244,-3.253,148.665,-165.122,117.838
C00374=-2.334,1.029,-3.254,153.984,-165.142,123.069
C00375=-2.422,0.806,-3.257,159.299,-165.195,128.330
C00376=-2.484,0.575,-3.260,164.626,-165.238,133.634
C00377=-2.526,0.340,-3.263,169.954,-165.291,138.974
C00378=-2.547,0.102,-3.265,175.289,-165.326,144.353
C00379=-2.545,-0.136,-3.266,-179.378,-165.350,149.762
C00380=-2.520,-0.374,-3.270,-174.043,-165.412,155.210
C00381=-2.473,-0.607,-3.273,-168.695,-165.440,160.694
C00382=-2.406,-0.836,-3.275,-163.348,-165.455,166.199
C00383=-2.317,-1.056,-3.277,-157.996,-165.474,171.725
C00384=-2.206,-1.267,-3.280,-152.641,-165.485,177.266
C00385=-2.079,-1.468,-3.284,-147.279,-165.500,-177.183
C00386=-1.932,-1.654,-3.285,-141.904,-165.474,-171.622
C00387=-1.769,-1.826,-3.287,-136.533,-165.456,-166.075
C00388=-1.591,-1.983,-3.290,-131.152,-165.437,-160.536
C00389=-1.399,-2.122,-3.293,-125.763,-165.399,-155.010
C00390=-1.195,-2.242,-3.296,-120.366,-165.375,-149.505
C00391=-0.981,-2.342,-3.297,-114.956,-165.317,-144.016
C00392=-0.760,-2.424,-3.300,-109.545,-165.274,-138.561
C00393=-0.532,-2.483,-3.304,-104.115,-165.244,-133.124
C00394=-0.299,-2.519,-3.306,-98.666,-165.194,-127.701
C00395=-0.066,-2.537,-3.308,-93.198,-165.150,-122.295
C00396=0.168,-2.531,-3.309,-87.702,-165.092,-116.891
C00397=0.514,-2.485,-3.315,-79.195,-165.071,-108.588
C00398=0.743,-2.423,-3.317,-73.856,-165.034,-103.402
C00399=0.967,-2.343,-3.318,-68.517,-165.012,-98.231
C00400=1.181,-2.242,-3.321,-63.171,-165.000,-93.064
C00401=1.385,-2.121,-3.324,-57.818,-165.006,-87.892
C00402=1.576,-1.982,-3.327,-52.451,-165.024,-82.705
C00403=1.753,-1.826,-3.328,-47.075,-165.019,-77.501
C00404=1.916,-1.655,-3.331,-41.695,-165.044,-72.279
C00405=2.060,-1.469,-3.335,-36.294,-165.092,-67.015
C00406=2.186,-1.270,-3.337,-30.877,-165.124,-61.712
C00407=2.296,-1.063,-3.339,-25.437,-165.164,-56.358
C00408=2.382,-0.846,-3.341,-19.970,-165.193,-50.946
C00409=2.471,-0.540,-3.346,-12.233,-165.284,-43.221
C00410=2.507,-0.305,-3.348,-6.959,-165.319,-37.916
C00411=2.528,-0.003,-3.350,0.000,-165.365,-30.867
C00412=2.513,0.235,-3.353,5.247,-165.405,-25.517
C00413=2.479,0.471,-3.357,10.503,-165.449,-20.129
C00414=2.425,0.703,-3.357,15.772,-165.465,-14.708
C00415=2.348,0.927,-3.356,21.045,-165.470,-9.266
C00416=2.250,1.144,-3.356,26.330,-165.496,-3.799
C00417=2.132,1.350,-3.357,31.634,-165.496,1.692
C00418=1.998,1.544,-3.357,36.954,-165.487,7.196
C00419=1.844,1.724,-3.356,42.300,-165.472,12.720
C00420=1.675,1.887,-3.356,47.675,-165.442,18.258
C00421=1.490,2.040,-3.357,53.385,-165.428,24.116
C00422=1.290,2.169,-3.357,58.665,-165.382,29.508
C00423=1.081,2.281,-3.356,63.941,-165.340,34.866
C00424=0.862,2.373,-3.356,69.220,-165.289,40.196
C00425=0.634,2.443,-3.357,74.498,-165.249,45.490
C00426=0.402,2.492,-3.357,79.782,-165.218,50.757
C00427=0.166,2.518,-3.356,85.071,-165.158,55.997
C00428=-0.071,2.524,-3.356,90.352,-165.106,61.200
C00429=-0.308,2.505,-3.357,95.641,-165.093,66.377
C00430=-0.542,2.464,-3.357,100.933,-165.058,71.538
C00431=-0.772,2.405,-3.357,106.227,-165.039,76.679
C00432=-0.993,2.320,-3.356,111.524,-165.001,81.809
C00433=-1.207,2.216,-3.356,116.817,-165.007,86.925
C00434=-1.410,2.094,-3.357,122.121,-165.009,92.049
C00435=-1.600,1.952,-3.356,127.425,-165.005,97.175
C00436=-1.776,1.794,-3.356,132.730,-165.023,102.310
C00437=-1.936,1.619,-3.356,138.038,-165.041,107.460
C00438=-2.080,1.431,-3.357,143.347,-165.074,112.632
C00439=-2.205,1.229,-3.357,148.665,-165.122,117.838
C00440=-2.309,1.017,-3.356,153.984,-165.142,123.069
C00441=-2.397,0.797,-3.356,159.299,-165.195,128.330
C00442=-2.459,0.568,-3.357,164.626,-165.238,133.634
C00443=-2.501,0.336,-3.357,169.954,-165.291,138.974
C00444=-2.523,0.100,-3.356,175.289,-165.326,144.353
C00445=-2.521,-0.136,-3.356,-179.378,-165.350,149.762
C00446=-2.497,-0.371,-3.357,-174.043,-165.412,155.210
C00447=-2.450,-0.603,-3.357,-168.695,-165.440,160.694
C00448=-2.385,-0.829,-3.356,-163.348,-165.455,166.199
C00449=-2.297,-1.048,-3.356,-157.996,-165.474,171.725
C00450=-2.187,-1.257,-3.357,-152.641,-165.485,177.266
C00451=-2.062,-1.457,-3.357,-147.279,-165.500,-177.183
C00452=-1.917,-1.642,-3.357,-141.904,-165.474,-171.622
C00453=-1.755,-1.814,-3.356,-136.533,-165.456,-166.075
C00454=-1.579,-1.970,-3.356,-131.152,-165.437,-160.536
C00455=-1.389,-2.108,-3.357,-125.763,-165.399,-155.010
C00456=-1.187,-2.228,-3.357,-120.366,-165.375,-149.505
C00457=-0.975,-2.328,-3.356,-114.956,-165.317,-144.016
C00458=-0.755,-2.409,-3.356,-109.545,-165.274,-138.561
C00459=-0.528,-2.469,-3.357,-104.115,-165.244,-133.124
C00460=-0.297,-2.505,-3.357,-98.666,-165.194,-127.701
C00461=-0.065,-2.524,-3.356,-93.198,-165.150,-122.295
C00462=0.168,-2.519,-3.356,-87.702,-165.092,-116.891
C00463=0.512,-2.474,-3.358,-79.195,-165.071,-108.588
C00464=0.740,-2.412,-3.357,-73.856,-165.034,-103.402
C00465=0.963,-2.333,-3.356,-68.517,-165.012,-98.231
C00466=1.177,-2.234,-3.356,-63.171,-165.000,-93.064
C00467=1.380,-2.113,-3.357,-57.818,-165.006,-87.892
C00468=1.571,-1.975,-3.357,-52.451,-165.024,-82.705
C00469=1.748,-1.820,-3.356,-47.075,-165.019,-77.501
C00470=1.911,-1.651,-3.356,-41.695,-165.044,-72.279
C00471=2.055,-1.465,-3.357,-36.294,-165.092,-67.015
C00472=2.182,-1.268,-3.357,-30.877,-165.124,-61.712
C00473=2.292,-1.061,-3.357,-25.437,-165.164,-56.358
C00474=2.378,-0.845,-3.356,-19.970,-165.193,-50.946
C00475=2.468,-0.540,-3.357,-12.233,-165.284,-43.221
C00476=2.505,-0.305,-3.357,-6.959,-165.319,-37.916
C00477=2.527,-0.003,-3.356,0.000,-165.365,-30.867
C00478=2.512,0.235,-3.356,5.247,-165.405,-25.517
C00479=2.479,0.471,-3.357,10.503,-165.449,-20.129
C00480=2.354,0.842,-3.347,12.864,-165.595,-17.690
C00481=2.161,1.182,-3.317,14.975,-165.947,-15.493
C00482=1.908,1.478,-3.269,16.598,-166.486,-13.790
C00483=1.605,1.718,-3.205,17.450,-167.179,-12.876
C00484=1.263,1.893,-3.126,17.184,-167.975,-13.106
C00485=0.895,1.996,-3.037,15.398,-168.796,-14.883
C00486=0.516,2.024,-2.940,11.418,-169.543,-18.883
C00487=0.141,1.975,-2.839,11.710,-170.143,-18.552
C00488=-0.236,1.927,-2.738,11.992,-170.738,-18.235
C00489=-0.578,1.883,-2.611,11.992,-170.738,-18.235
C00490=-0.892,1.844,-2.423,11.992,-170.738,-18.235
C00491=-1.167,1.811,-2.180,11.992,-170.738,-18.235
C00492=-1.393,1.785,-1.891,11.992,-170.738,-18.235
C00493=-1.562,1.767,-1.565,11.992,-170.738,-18.235
C00494=-1.670,1.757,-1.213,11.992,-170.738,-18.235
C00495=-1.712,1.756,-0.848,11.992,-170.738,-18.235
C00496=-1.686,1.764,-0.481,11.992,-170.738,-18.235
C00497=-1.397,1.826,1.312,11.992,-170.738,-18.235
C00498=-1.397,1.826,16.000,11.992,-170.738,-18.235
//INST
///ATTR SC,RW,RJ
////FRAME USER 1
///GROUP1 RB1
///LVARS 2,0,0,0,0,0,0,0
NOP
SET LB000 1
SET LB001 25
MOVJ C00000 VJ=17
MOVL C00001 V=17 PL=LB000 ACC=LB001 DEC=LB001
' Lead In Move Starts
MOVL C00002 V=17 PL=LB000 ACC=LB001 DEC=LB001
' Cutting Move Starts
MOVL C00003 V=17 PL=LB000 ACC=LB001 DEC=LB001
MOVL C00004 V=17 PL=LB000 ACC=LB001 DEC=LB001
MOVL C00005 V=17 PL=LB000 ACC=LB001 DEC=LB001
MOVL C00006 V=17 PL=LB000 ACC=LB001 DEC=LB001
MOVL C00007 V=17 PL=LB000 ACC=LB001 DEC=LB001
MOVL C00008 V=17 PL=LB000 ACC=LB001 DEC=LB001
MOVL C00009 V=17 PL=LB000 ACC=LB001 DEC=LB001
MOVL C00010 V=17 PL=LB000 ACC=LB001 DEC=LB001
MOVL C00011 V=17 PL=LB000 ACC=LB001 DEC=LB001
MOVL C00012 V=17 PL=LB000 ACC=LB001 DEC=LB001
MOVL C00013 V=17 PL=LB000 ACC=LB001 DEC=LB001
MOVL C00014 V=17 PL=LB000 ACC=LB001 DEC=LB001
MOVL C00015 V=17 PL=LB000 ACC=LB001 DEC=LB001
MOVL C00016 V=17 PL=LB000 ACC=LB001 DEC=LB001
MOVL C00017 V=17 PL=LB000 ACC=LB001 DEC=LB001
MOVL C00018 V=17 PL=LB000 ACC=LB001 DEC=LB001
MOVL C00019 V=17 PL=LB000 ACC=LB001 DEC=LB001
MOVL C00020 V=17 PL=LB000 ACC=LB001 DEC=LB001
MOVL C00021 V=17 PL=LB000 ACC=LB001 DEC=LB001
MOVL C00022 V=17 PL=LB000 ACC=LB001 DEC=LB001
MOVL C00023 V=17 PL=LB000 ACC=LB001 DEC=LB001
MOVL C00024 V=17 PL=LB000 ACC=LB001 DEC=LB001
MOVL C00025 V=17 PL=LB000 ACC=LB001 DEC=LB001
MOVL C00026 V=17 PL=LB000 ACC=LB001 DEC=LB001
' Lead Out Move Starts
MOVL C00027 V=17 PL=LB000 ACC=LB001 DEC=LB001
' Rapid Move Starts
MOVL C00028 V=17 PL=LB000 ACC=LB001 DEC=LB001
' By Autodesk Fusion CAM 2.0.20494
' Tool = 8
' Spindle = 6000 RPM
' Set Position Level
' Set Acceleration
' Program Start
' First Toolpath Point
' Last Toolpath Point
MOVJ C00000 VJ=17
MOVL C00001 V=17 PL=LB000 ACC=LB001 DEC=LB001
' Plunge Move Starts
MOVL C00002 V=8 PL=LB000 ACC=LB001 DEC=LB001
' Lead In Move Starts
MOVL C00003 V=17 PL=LB000 ACC=LB001 DEC=LB001
MOVL C00004 V=17 PL=LB000 ACC=LB001 DEC=LB001
' Cutting Move Starts
MOVL C00005 V=17 PL=LB000 ACC=LB001 DEC=LB001
' Lead Out Move Starts
MOVL C00006 V=17 PL=LB000 ACC=LB001 DEC=LB001
MOVL C00007 V=17 PL=LB000 ACC=LB001 DEC=LB001
' Rapid Move Starts
MOVL C00008 V=17 PL=LB000 ACC=LB001 DEC=LB001
' By Autodesk Fusion CAM 2.0.20494
' Tool = 2
' Spindle = 5000 RPM
' Set Position Level
' Set Acceleration
' Program Start
' First Toolpath Point
' Last Toolpath Point
MOVJ C00000 VJ=17
MOVL C00001 V=17 PL=LB000 ACC=LB001 DEC=LB001
' Lead In Move Starts
MOVL C00002 V=17 PL=LB000 ACC=LB001 DEC=LB001
' Cutting Move Starts
MOVL C00003 V=17 PL=LB000 ACC=LB001 DEC=LB001
MOVL C00004 V=17 PL=LB000 ACC=LB001 DEC=LB001
MOVL C00005 V=17 PL=LB000 ACC=LB001 DEC=LB001
MOVL C00006 V=17 PL=LB000 ACC=LB001 DEC=LB001
MOVL C00007 V=17 PL=LB000 ACC=LB001 DEC=LB001
MOVL C00008 V=17 PL=LB000 ACC=LB001 DEC=LB001
MOVL C00009 V=17 PL=LB000 ACC=LB001 DEC=LB001
MOVL C00010 V=17 PL=LB000 ACC=LB001 DEC=LB001
MOVL C00011 V=17 PL=LB000 ACC=LB001 DEC=LB001
MOVL C00012 V=17 PL=LB000 ACC=LB001 DEC=LB001
MOVL C00013 V=17 PL=LB000 ACC=LB001 DEC=LB001
MOVL C00014 V=17 PL=LB000 ACC=LB001 DEC=LB001
MOVL C00015 V=17 PL=LB000 ACC=LB001 DEC=LB001
MOVL C00016 V=17 PL=LB000 ACC=LB001 DEC=LB001
MOVL C00017 V=17 PL=LB000 ACC=LB001 DEC=LB001
' Lead Out Move Starts
MOVL C00018 V=17 PL=LB000 ACC=LB001 DEC=LB001
' Rapid Move Starts
MOVL C00019 V=17 PL=LB000 ACC=LB001 DEC=LB001
' By Autodesk Fusion CAM 2.0.20494
' Tool = 8
' Spindle = 6000 RPM
' Set Position Level
' Set Acceleration
' Program Start
' First Toolpath Point
' Last Toolpath Point
MOVJ C00000 VJ=17
MOVL C00001 V=17 PL=LB000 ACC=LB001 DEC=LB001
' Plunge Move Starts
MOVL C00002 V=8 PL=LB000 ACC=LB001 DEC=LB001
' Lead In Move Starts
MOVL C00003 V=17 PL=LB000 ACC=LB001 DEC=LB001
MOVL C00004 V=17 PL=LB000 ACC=LB001 DEC=LB001
' Cutting Move Starts
MOVL C00005 V=17 PL=LB000 ACC=LB001 DEC=LB001
' Lead Out Move Starts
MOVL C00006 V=17 PL=LB000 ACC=LB001 DEC=LB001
MOVL C00007 V=17 PL=LB000 ACC=LB001 DEC=LB001
' Rapid Move Starts
MOVL C00008 V=17 PL=LB000 ACC=LB001 DEC=LB001
' By Autodesk Fusion CAM 2.0.20494
' Tool = 8
' Spindle = 6000 RPM
' Set Position Level
' Set Acceleration
' Program Start
' First Toolpath Point
' Last Toolpath Point
MOVJ C00000 VJ=17
MOVL C00001 V=17 PL=LB000 ACC=LB001 DEC=LB001
' Lead In Move Starts
MOVL C00002 V=17 PL=LB000 ACC=LB001 DEC=LB001
' Cutting Move Starts
MOVL C00003 V=17 PL=LB000 ACC=LB001 DEC=LB001
MOVL C00004 V=17 PL=LB000 ACC=LB001 DEC=LB001
MOVL C00005 V=17 PL=LB000 ACC=LB001 DEC=LB001
MOVL C00006 V=17 PL=LB000 ACC=LB001 DEC=LB001
MOVL C00007 V=17 PL=LB000 ACC=LB001 DEC=LB001
MOVL C00008 V=17 PL=LB000 ACC=LB001 DEC=LB001
MOVL C00009 V=17 PL=LB000 ACC=LB001 DEC=LB001
MOVL C00010 V=17 PL=LB000 ACC=LB001 DEC=LB001
MOVL C00011 V=17 PL=LB000 ACC=LB001 DEC=LB001
MOVL C00012 V=17 PL=LB000 ACC=LB001 DEC=LB001
MOVL C00013 V=17 PL=LB000 ACC=LB001 DEC=LB001
MOVL C00014 V=17 PL=LB000 ACC=LB001 DEC=LB001
MOVL C00015 V=17 PL=LB000 ACC=LB001 DEC=LB001
MOVL C00016 V=17 PL=LB000 ACC=LB001 DEC=LB001
MOVL C00017 V=17 PL=LB000 ACC=LB001 DEC=LB001
MOVL C00018 V=17 PL=LB000 ACC=LB001 DEC=LB001
MOVL C00019 V=17 PL=LB000 ACC=LB001 DEC=LB001
MOVL C00020 V=17 PL=LB000 ACC=LB001 DEC=LB001
MOVL C00021 V=17 PL=LB000 ACC=LB001 DEC=LB001
MOVL C00022 V=17 PL=LB000 ACC=LB001 DEC=LB001
MOVL C00023 V=17 PL=LB000 ACC=LB001 DEC=LB001
MOVL C00024 V=17 PL=LB000 ACC=LB001 DEC=LB001
MOVL C00025 V=17 PL=LB000 ACC=LB001 DEC=LB001
MOVL C00026 V=17 PL=LB000 ACC=LB001 DEC=LB001
' Lead Out Move Starts
MOVL C00027 V=17 PL=LB000 ACC=LB001 DEC=LB001
' Rapid Move Starts
MOVL C00028 V=17 PL=LB000 ACC=LB001 DEC=LB001
' By Autodesk Fusion CAM 2.0.20494
' Tool = 8
' Spindle = 6000 RPM
' Set Position Level
' Set Acceleration
' Program Start
' First Toolpath Point
' Last Toolpath Point
MOVJ C00000 VJ=17
MOVL C00001 V=17 PL=LB000 ACC=LB001 DEC=LB001
' Lead In Move Starts
MOVL C00002 V=17 PL=LB000 ACC=LB001 DEC=LB001
' Cutting Move Starts
MOVL C00003 V=17 PL=LB000 ACC=LB001 DEC=LB001
MOVL C00004 V=17 PL=LB000 ACC=LB001 DEC=LB001
MOVL C00005 V=17 PL=LB000 ACC=LB001 DEC=LB001
MOVL C00006 V=17 PL=LB000 ACC=LB001 DEC=LB001
MOVL C00007 V=17 PL=LB000 ACC=LB001 DEC=LB001
MOVL C00008 V=17 PL=LB000 ACC=LB001 DEC=LB001
MOVL C00009 V=17 PL=LB000 ACC=LB001 DEC=LB001
MOVL C00010 V=17 PL=LB000 ACC=LB001 DEC=LB001
MOVL C00011 V=17 PL=LB000 ACC=LB001 DEC=LB001
MOVL C00012 V=17 PL=LB000 ACC=LB001 DEC=LB001
MOVL C00013 V=17 PL=LB000 ACC=LB001 DEC=LB001
MOVL C00014 V=17 PL=LB000 ACC=LB001 DEC=LB001
MOVL C00015 V=17 PL=LB000 ACC=LB001 DEC=LB001
MOVL C00016 V=17 PL=LB000 ACC=LB001 DEC=LB001
MOVL C00017 V=17 PL=LB000 ACC=LB001 DEC=LB001
MOVL C00018 V=17 PL=LB000 ACC=LB001 DEC=LB001
MOVL C00019 V=17 PL=LB000 ACC=LB001 DEC=LB001
MOVL C00020 V=17 PL=LB000 ACC=LB001 DEC=LB001
MOVL C00021 V=17 PL=LB000 ACC=LB001 DEC=LB001
MOVL C00022 V=17 PL=LB000 ACC=LB001 DEC=LB001
MOVL C00023 V=17 PL=LB000 ACC=LB001 DEC=LB001
MOVL C00024 V=17 PL=LB000 ACC=LB001 DEC=LB001
MOVL C00025 V=17 PL=LB000 ACC=LB001 DEC=LB001
MOVL C00026 V=17 PL=LB000 ACC=LB001 DEC=LB001
' Lead Out Move Starts
MOVL C00027 V=17 PL=LB000 ACC=LB001 DEC=LB001
' Rapid Move Starts
MOVL C00028 V=17 PL=LB000 ACC=LB001 DEC=LB001
' By Autodesk Fusion CAM 2.0.20494
' Tool = 8
' Spindle = 6000 RPM
' Set Position Level
' Set Acceleration
' Program Start
' First Toolpath Point
' Last Toolpath Point
MOVJ C00000 VJ=17
MOVL C00001 V=17 PL=LB000 ACC=LB001 DEC=LB001
' Lead In Move Starts
MOVL C00002 V=17 PL=LB000 ACC=LB001 DEC=LB001
' Cutting Move Starts
MOVL C00003 V=17 PL=LB000 ACC=LB001 DEC=LB001
MOVL C00004 V=17 PL=LB000 ACC=LB001 DEC=LB001
MOVL C00005 V=17 PL=LB000 ACC=LB001 DEC=LB001
MOVL C00006 V=17 PL=LB000 ACC=LB001 DEC=LB001
MOVL C00007 V=17 PL=LB000 ACC=LB001 DEC=LB001
MOVL C00008 V=17 PL=LB000 ACC=LB001 DEC=LB001
MOVL C00009 V=17 PL=LB000 ACC=LB001 DEC=LB001
MOVL C00010 V=17 PL=LB000 ACC=LB001 DEC=LB001
MOVL C00011 V=17 PL=LB000 ACC=LB001 DEC=LB001
MOVL C00012 V=17 PL=LB000 ACC=LB001 DEC=LB001
MOVL C00013 V=17 PL=LB000 ACC=LB001 DEC=LB001
MOVL C00014 V=17 PL=LB000 ACC=LB001 DEC=LB001
MOVL C00015 V=17 PL=LB000 ACC=LB001 DEC=LB001
' Lead Out Move Starts
MOVL C00016 V=17 PL=LB000 ACC=LB001 DEC=LB001
' Rapid Move Starts
MOVL C00017 V=17 PL=LB000 ACC=LB001 DEC=LB001
' By Autodesk Fusion CAM 2.0.20494
' Tool = 8
' Spindle = 6000 RPM
' Set Position Level
' Set Acceleration
' Program Start
' First Toolpath Point
' Last Toolpath Point
MOVJ C00000 VJ=17
MOVL C00001 V=17 PL=LB000 ACC=LB001 DEC=LB001
' Lead In Move Starts
MOVL C00002 V=17 PL=LB000 ACC=LB001 DEC=LB001
' Cutting Move Starts
MOVL C00003 V=17 PL=LB000 ACC=LB001 DEC=LB001
MOVL C00004 V=17 PL=LB000 ACC=LB001 DEC=LB001
MOVL C00005 V=17 PL=LB000 ACC=LB001 DEC=LB001
MOVL C00006 V=17 PL=LB000 ACC=LB001 DEC=LB001
MOVL C00007 V=17 PL=LB000 ACC=LB001 DEC=LB001
MOVL C00008 V=17 PL=LB000 ACC=LB001 DEC=LB001
MOVL C00009 V=17 PL=LB000 ACC=LB001 DEC=LB001
MOVL C00010 V=17 PL=LB000 ACC=LB001 DEC=LB001
MOVL C00011 V=17 PL=LB000 ACC=LB001 DEC=LB001
MOVL C00012 V=17 PL=LB000 ACC=LB001 DEC=LB001
MOVL C00013 V=17 PL=LB000 ACC=LB001 DEC=LB001
MOVL C00014 V=17 PL=LB000 ACC=LB001 DEC=LB001
' Lead Out Move Starts
MOVL C00015 V=17 PL=LB000 ACC=LB001 DEC=LB001
' Rapid Move Starts
MOVL C00016 V=17 PL=LB000 ACC=LB001 DEC=LB001
' By Autodesk Fusion CAM 2.0.20494
' Tool = 2
' Spindle = 5000 RPM
' Set Position Level
' Set Acceleration
' Program Start
' First Toolpath Point
' Last Toolpath Point
MOVJ C00000 VJ=17
MOVL C00001 V=17 PL=LB000 ACC=LB001 DEC=LB001
' Lead In Move Starts
MOVL C00002 V=17 PL=LB000 ACC=LB001 DEC=LB001
' Cutting Move Starts
MOVL C00003 V=17 PL=LB000 ACC=LB001 DEC=LB001
MOVL C00004 V=17 PL=LB000 ACC=LB001 DEC=LB001
MOVL C00005 V=17 PL=LB000 ACC=LB001 DEC=LB001
MOVL C00006 V=17 PL=LB000 ACC=LB001 DEC=LB001
' Lead Out Move Starts
MOVL C00007 V=17 PL=LB000 ACC=LB001 DEC=LB001
' Rapid Move Starts
MOVL C00008 V=17 PL=LB000 ACC=LB001 DEC=LB001
MOVL C00009 V=17 PL=LB000 ACC=LB001 DEC=LB001
' By Autodesk Fusion CAM 2.0.20494
' Tool = 8
' Spindle = 6000 RPM
' Set Position Level
' Set Acceleration
' Program Start
' First Toolpath Point
' Last Toolpath Point
MOVJ C00000 VJ=17
MOVL C00001 V=17 PL=LB000 ACC=LB001 DEC=LB001
' Plunge Move Starts
MOVL C00002 V=8 PL=LB000 ACC=LB001 DEC=LB001
MOVL C00003 V=8 PL=LB000 ACC=LB001 DEC=LB001
' Lead In Move Starts
MOVL C00004 V=17 PL=LB000 ACC=LB001 DEC=LB001
MOVL C00005 V=17 PL=LB000 ACC=LB001 DEC=LB001
MOVL C00006 V=17 PL=LB000 ACC=LB001 DEC=LB001
MOVL C00007 V=17 PL=LB000 ACC=LB001 DEC=LB001
MOVL C00008 V=17 PL=LB000 ACC=LB001 DEC=LB001
' Cutting Move Starts
MOVL C00009 V=17 PL=LB000 ACC=LB001 DEC=LB001
MOVL C00010 V=17 PL=LB000 ACC=LB001 DEC=LB001
MOVL C00011 V=17 PL=LB000 ACC=LB001 DEC=LB001
MOVL C00012 V=17 PL=LB000 ACC=LB001 DEC=LB001
MOVL C00013 V=17 PL=LB000 ACC=LB001 DEC=LB001
MOVL C00014 V=17 PL=LB000 ACC=LB001 DEC=LB001
MOVL C00015 V=17 PL=LB000 ACC=LB001 DEC=LB001
MOVL C00016 V=17 PL=LB000 ACC=LB001 DEC=LB001
MOVL C00017 V=17 PL=LB000 ACC=LB001 DEC=LB001
MOVL C00018 V=17 PL=LB000 ACC=LB001 DEC=LB001
MOVL C00019 V=17 PL=LB000 ACC=LB001 DEC=LB001
' Lead Out Move Starts
MOVL C00020 V=17 PL=LB000 ACC=LB001 DEC=LB001
MOVL C00021 V=17 PL=LB000 ACC=LB001 DEC=LB001
MOVL C00022 V=17 PL=LB000 ACC=LB001 DEC=LB001
MOVL C00023 V=17 PL=LB000 ACC=LB001 DEC=LB001
MOVL C00024 V=17 PL=LB000 ACC=LB001 DEC=LB001
' Rapid Move Starts
MOVL C00025 V=17 PL=LB000 ACC=LB001 DEC=LB001
' By Autodesk Fusion CAM 2.0.20494
' Tool = 8
' Spindle = 6000 RPM
' Set Position Level
' Set Acceleration
' Program Start
' First Toolpath Point
' Last Toolpath Point
MOVJ C00000 VJ=17
MOVL C00001 V=17 PL=LB000 ACC=LB001 DEC=LB001
' Lead In Move Starts
MOVL C00002 V=17 PL=LB000 ACC=LB001 DEC=LB001
MOVL C00003 V=17 PL=LB000 ACC=LB001 DEC=LB001
MOVL C00004 V=17 PL=LB000 ACC=LB001 DEC=LB001
MOVL C00005 V=17 PL=LB000 ACC=LB001 DEC=LB001
MOVL C00006 V=17 PL=LB000 ACC=LB001 DEC=LB001
MOVL C00007 V=17 PL=LB000 ACC=LB001 DEC=LB001
MOVL C00008 V=17 PL=LB000 ACC=LB001 DEC=LB001
MOVL C00009 V=17 PL=LB000 ACC=LB001 DEC=LB001
MOVL C00010 V=17 PL=LB000 ACC=LB001 DEC=LB001
MOVL C00011 V=17 PL=LB000 ACC=LB001 DEC=LB001
MOVL C00012 V=17 PL=LB000 ACC=LB001 DEC=LB001
MOVL C00013 V=17 PL=LB000 ACC=LB001 DEC=LB001
MOVL C00014 V=17 PL=LB000 ACC=LB001 DEC=LB001
MOVL C00015 V=17 PL=LB000 ACC=LB001 DEC=LB001
MOVL C00016 V=17 PL=LB000 ACC=LB001 DEC=LB001
MOVL C00017 V=17 PL=LB000 ACC=LB001 DEC=LB001
' Cutting Move Starts
MOVL C00018 V=17 PL=LB000 ACC=LB001 DEC=LB001
MOVL C00019 V=17 PL=LB000 ACC=LB001 DEC=LB001
MOVL C00020 V=17 PL=LB000 ACC=LB001 DEC=LB001
MOVL C00021 V=17 PL=LB000 ACC=LB001 DEC=LB001
MOVL C00022 V=17 PL=LB000 ACC=LB001 DEC=LB001
MOVL C00023 V=17 PL=LB000 ACC=LB001 DEC=LB001
MOVL C00024 V=17 PL=LB000 ACC=LB001 DEC=LB001
MOVL C00025 V=17 PL=LB000 ACC=LB001 DEC=LB001
MOVL C00026 V=17 PL=LB000 ACC=LB001 DEC=LB001
MOVL C00027 V=17 PL=LB000 ACC=LB001 DEC=LB001
MOVL C00028 V=17 PL=LB000 ACC=LB001 DEC=LB001
MOVL C00029 V=17 PL=LB000 ACC=LB001 DEC=LB001
MOVL C00030 V=17 PL=LB000 ACC=LB001 DEC=LB001
MOVL C00031 V=17 PL=LB000 ACC=LB001 DEC=LB001
MOVL C00032 V=17 PL=LB000 ACC=LB001 DEC=LB001
MOVL C00033 V=17 PL=LB000 ACC=LB001 DEC=LB001
MOVL C00034 V=17 PL=LB000 ACC=LB001 DEC=LB001
MOVL C00035 V=17 PL=LB000 ACC=LB001 DEC=LB001
MOVL C00036 V=17 PL=LB000 ACC=LB001 DEC=LB001
MOVL C00037 V=17 PL=LB000 ACC=LB001 DEC=LB001
MOVL C00038 V=17 PL=LB000 ACC=LB001 DEC=LB001
MOVL C00039 V=17 PL=LB000 ACC=LB001 DEC=LB001
MOVL C00040 V=17 PL=LB000 ACC=LB001 DEC=LB001
MOVL C00041 V=17 PL=LB000 ACC=LB001 DEC=LB001
MOVL C00042 V=17 PL=LB000 ACC=LB001 DEC=LB001
MOVL C00043 V=17 PL=LB000 ACC=LB001 DEC=LB001
MOVL C00044 V=17 PL=LB000 ACC=LB001 DEC=LB001
MOVL C00045 V=17 PL=LB000 ACC=LB001 DEC=LB001
MOVL C00046 V=17 PL=LB000 ACC=LB001 DEC=LB001
MOVL C00047 V=17 PL=LB000 ACC=LB001 DEC=LB001
MOVL C00048 V=17 PL=LB000 ACC=LB001 DEC=LB001
MOVL C00049 V=17 PL=LB000 ACC=LB001 DEC=LB001
MOVL C00050 V=17 PL=LB000 ACC=LB001 DEC=LB001
MOVL C00051 V=17 PL=LB000 ACC=LB001 DEC=LB001
MOVL C00052 V=17 PL=LB000 ACC=LB001 DEC=LB001
MOVL C00053 V=17 PL=LB000 ACC=LB001 DEC=LB001
MOVL C00054 V=17 PL=LB000 ACC=LB001 DEC=LB001
MOVL C00055 V=17 PL=LB000 ACC=LB001 DEC=LB001
MOVL C00056 V=17 PL=LB000 ACC=LB001 DEC=LB001
MOVL C00057 V=17 PL=LB000 ACC=LB001 DEC=LB001
MOVL C00058 V=17 PL=LB000 ACC=LB001 DEC=LB001
MOVL C00059 V=17 PL=LB000 ACC=LB001 DEC=LB001
MOVL C00060 V=17 PL=LB000 ACC=LB001 DEC=LB001
MOVL C00061 V=17 PL=LB000 ACC=LB001 DEC=LB001
MOVL C00062 V=17 PL=LB000 ACC=LB001 DEC=LB001
MOVL C00063 V=17 PL=LB000 ACC=LB001 DEC=LB001
MOVL C00064 V=17 PL=LB000 ACC=LB001 DEC=LB001
MOVL C00065 V=17 PL=LB000 ACC=LB001 DEC=LB001
MOVL C00066 V=17 PL=LB000 ACC=LB001 DEC=LB001
MOVL C00067 V=17 PL=LB000 ACC=LB001 DEC=LB001
MOVL C00068 V=17 PL=LB000 ACC=LB001 DEC=LB001
MOVL C00069 V=17 PL=LB000 ACC=LB001 DEC=LB001
MOVL C00070 V=17 PL=LB000 ACC=LB001 DEC=LB001
MOVL C00071 V=17 PL=LB000 ACC=LB001 DEC=LB001
MOVL C00072 V=17 PL=LB000 ACC=LB001 DEC=LB001
MOVL C00073 V=17 PL=LB000 ACC=LB001 DEC=LB001
MOVL C00074 V=17 PL=LB000 ACC=LB001 DEC=LB001
MOVL C00075 V=17 PL=LB000 ACC=LB001 DEC=LB001
MOVL C00076 V=17 PL=LB000 ACC=LB001 DEC=LB001
MOVL C00077 V=17 PL=LB000 ACC=LB001 DEC=LB001
MOVL C00078 V=17 PL=LB000 ACC=LB001 DEC=LB001
MOVL C00079 V=17 PL=LB000 ACC=LB001 DEC=LB001
MOVL C00080 V=17 PL=LB000 ACC=LB001 DEC=LB001
MOVL C00081 V=17 PL=LB000 ACC=LB001 DEC=LB001
MOVL C00082 V=17 PL=LB000 ACC=LB001 DEC=LB001
MOVL C00083 V=17 PL=LB000 ACC=LB001 DEC=LB001
MOVL C00084 V=17 PL=LB000 ACC=LB001 DEC=LB001
MOVL C00085 V=17 PL=LB000 ACC=LB001 DEC=LB001
MOVL C00086 V=17 PL=LB000 ACC=LB001 DEC=LB001
MOVL C00087 V=17 PL=LB000 ACC=LB001 DEC=LB001
MOVL C00088 V=17 PL=LB000 ACC=LB001 DEC=LB001
MOVL C00089 V=17 PL=LB000 ACC=LB001 DEC=LB001
MOVL C00090 V=17 PL=LB000 ACC=LB001 DEC=LB001
MOVL C00091 V=17 PL=LB000 ACC=LB001 DEC=LB001
MOVL C00092 V=17 PL=LB000 ACC=LB001 DEC=LB001
MOVL C00093 V=17 PL=LB000 ACC=LB001 DEC=LB001
MOVL C00094 V=17 PL=LB000 ACC=LB001 DEC=LB001
MOVL C00095 V=17 PL=LB000 ACC=LB001 DEC=LB001
MOVL C00096 V=17 PL=LB000 ACC=LB001 DEC=LB001
MOVL C00097 V=17 PL=LB000 ACC=LB001 DEC=LB001
MOVL C00098 V=17 PL=LB000 ACC=LB001 DEC=LB001
MOVL C00099 V=17 PL=LB000 ACC=LB001 DEC=LB001
MOVL C00100 V=17 PL=LB000 ACC=LB001 DEC=LB001
MOVL C00101 V=17 PL=LB000 ACC=LB001 DEC=LB001
MOVL C00102 V=17 PL=LB000 ACC=LB001 DEC=LB001
MOVL C00103 V=17 PL=LB000 ACC=LB001 DEC=LB001
MOVL C00104 V=17 PL=LB000 ACC=LB001 DEC=LB001
MOVL C00105 V=17 PL=LB000 ACC=LB001 DEC=LB001
MOVL C00106 V=17 PL=LB000 ACC=LB001 DEC=LB001
MOVL C00107 V=17 PL=LB000 ACC=LB001 DEC=LB001
MOVL C00108 V=17 PL=LB000 ACC=LB001 DEC=LB001
MOVL C00109 V=17 PL=LB000 ACC=LB001 DEC=LB001
MOVL C00110 V=17 PL=LB000 ACC=LB001 DEC=LB001
MOVL C00111 V=17 PL=LB000 ACC=LB001 DEC=LB001
MOVL C00112 V=17 PL=LB000 ACC=LB001 DEC=LB001
MOVL C00113 V=17 PL=LB000 ACC=LB001 DEC=LB001
MOVL C00114 V=17 PL=LB000 ACC=LB001 DEC=LB001
MOVL C00115 V=17 PL=LB000 ACC=LB001 DEC=LB001
MOVL C00116 V=17 PL=LB000 ACC=LB001 DEC=LB001
MOVL C00117 V=17 PL=LB000 ACC=LB001 DEC=LB001
MOVL C00118 V=17 PL=LB000 ACC=LB001 DEC=LB001
MOVL C00119 V=17 PL=LB000 ACC=LB001 DEC=LB001
MOVL C00120 V=17 PL=LB000 ACC=LB001 DEC=LB001
MOVL C00121 V=17 PL=LB000 ACC=LB001 DEC=LB001
MOVL C00122 V=17 PL=LB000 ACC=LB001 DEC=LB001
MOVL C00123 V=17 PL=LB000 ACC=LB001 DEC=LB001
MOVL C00124 V=17 PL=LB000 ACC=LB001 DEC=LB001
MOVL C00125 V=17 PL=LB000 ACC=LB001 DEC=LB001
MOVL C00126 V=17 PL=LB000 ACC=LB001 DEC=LB001
MOVL C00127 V=17 PL=LB000 ACC=LB001 DEC=LB001
MOVL C00128 V=17 PL=LB000 ACC=LB001 DEC=LB001
MOVL C00129 V=17 PL=LB000 ACC=LB001 DEC=LB001
MOVL C00130 V=17 PL=LB000 ACC=LB001 DEC=LB001
MOVL C00131 V=17 PL=LB000 ACC=LB001 DEC=LB001
MOVL C00132 V=17 PL=LB000 ACC=LB001 DEC=LB001
MOVL C00133 V=17 PL=LB000 ACC=LB001 DEC=LB001
MOVL C00134 V=17 PL=LB000 ACC=LB001 DEC=LB001
MOVL C00135 V=17 PL=LB000 ACC=LB001 DEC=LB001
MOVL C00136 V=17 PL=LB000 ACC=LB001 DEC=LB001
MOVL C00137 V=17 PL=LB000 ACC=LB001 DEC=LB001
MOVL C00138 V=17 PL=LB000 ACC=LB001 DEC=LB001
MOVL C00139 V=17 PL=LB000 ACC=LB001 DEC=LB001
MOVL C00140 V=17 PL=LB000 ACC=LB001 DEC=LB001
MOVL C00141 V=17 PL=LB000 ACC=LB001 DEC=LB001
MOVL C00142 V=17 PL=LB000 ACC=LB001 DEC=LB001
MOVL C00143 V=17 PL=LB000 ACC=LB001 DEC=LB001
MOVL C00144 V=17 PL=LB000 ACC=LB001 DEC=LB001
MOVL C00145 V=17 PL=LB000 ACC=LB001 DEC=LB001
MOVL C00146 V=17 PL=LB000 ACC=LB001 DEC=LB001
MOVL C00147 V=17 PL=LB000 ACC=LB001 DEC=LB001
MOVL C00148 V=17 PL=LB000 ACC=LB001 DEC=LB001
MOVL C00149 V=17 PL=LB000 ACC=LB001 DEC=LB001
MOVL C00150 V=17 PL=LB000 ACC=LB001 DEC=LB001
MOVL C00151 V=17 PL=LB000 ACC=LB001 DEC=LB001
MOVL C00152 V=17 PL=LB000 ACC=LB001 DEC=LB001
MOVL C00153 V=17 PL=LB000 ACC=LB001 DEC=LB001
MOVL C00154 V=17 PL=LB000 ACC=LB001 DEC=LB001
MOVL C00155 V=17 PL=LB000 ACC=LB001 DEC=LB001
MOVL C00156 V=17 PL=LB000 ACC=LB001 DEC=LB001
MOVL C00157 V=17 PL=LB000 ACC=LB001 DEC=LB001
MOVL C00158 V=17 PL=LB000 ACC=LB001 DEC=LB001
MOVL C00159 V=17 PL=LB000 ACC=LB001 DEC=LB001
MOVL C00160 V=17 PL=LB000 ACC=LB001 DEC=LB001
MOVL C00161 V=17 PL=LB000 ACC=LB001 DEC=LB001
MOVL C00162 V=17 PL=LB000 ACC=LB001 DEC=LB001
MOVL C00163 V=17 PL=LB000 ACC=LB001 DEC=LB001
MOVL C00164 V=17 PL=LB000 ACC=LB001 DEC=LB001
MOVL C00165 V=17 PL=LB000 ACC=LB001 DEC=LB001
MOVL C00166 V=17 PL=LB000 ACC=LB001 DEC=LB001
MOVL C00167 V=17 PL=LB000 ACC=LB001 DEC=LB001
MOVL C00168 V=17 PL=LB000 ACC=LB001 DEC=LB001
MOVL C00169 V=17 PL=LB000 ACC=LB001 DEC=LB001
MOVL C00170 V=17 PL=LB000 ACC=LB001 DEC=LB001
MOVL C00171 V=17 PL=LB000 ACC=LB001 DEC=LB001
MOVL C00172 V=17 PL=LB000 ACC=LB001 DEC=LB001
MOVL C00173 V=17 PL=LB000 ACC=LB001 DEC=LB001
MOVL C00174 V=17 PL=LB000 ACC=LB001 DEC=LB001
MOVL C00175 V=17 PL=LB000 ACC=LB001 DEC=LB001
MOVL C00176 V=17 PL=LB000 ACC=LB001 DEC=LB001
MOVL C00177 V=17 PL=LB000 ACC=LB001 DEC=LB001
MOVL C00178 V=17 PL=LB000 ACC=LB001 DEC=LB001
MOVL C00179 V=17 PL=LB000 ACC=LB001 DEC=LB001
MOVL C00180 V=17 PL=LB000 ACC=LB001 DEC=LB001
MOVL C00181 V=17 PL=LB000 ACC=LB001 DEC=LB001
MOVL C00182 V=17 PL=LB000 ACC=LB001 DEC=LB001
MOVL C00183 V=17 PL=LB000 ACC=LB001 DEC=LB001
MOVL C00184 V=17 PL=LB000 ACC=LB001 DEC=LB001
MOVL C00185 V=17 PL=LB000 ACC=LB001 DEC=LB001
MOVL C00186 V=17 PL=LB000 ACC=LB001 DEC=LB001
MOVL C00187 V=17 PL=LB000 ACC=LB001 DEC=LB001
MOVL C00188 V=17 PL=LB000 ACC=LB001 DEC=LB001
MOVL C00189 V=17 PL=LB000 ACC=LB001 DEC=LB001
MOVL C00190 V=17 PL=LB000 ACC=LB001 DEC=LB001
MOVL C00191 V=17 PL=LB000 ACC=LB001 DEC=LB001
MOVL C00192 V=17 PL=LB000 ACC=LB001 DEC=LB001
MOVL C00193 V=17 PL=LB000 ACC=LB001 DEC=LB001
MOVL C00194 V=17 PL=LB000 ACC=LB001 DEC=LB001
MOVL C00195 V=17 PL=LB000 ACC=LB001 DEC=LB001
MOVL C00196 V=17 PL=LB000 ACC=LB001 DEC=LB001
MOVL C00197 V=17 PL=LB000 ACC=LB001 DEC=LB001
MOVL C00198 V=17 PL=LB000 ACC=LB001 DEC=LB001
MOVL C00199 V=17 PL=LB000 ACC=LB001 DEC=LB001
MOVL C00200 V=17 PL=LB000 ACC=LB001 DEC=LB001
MOVL C00201 V=17 PL=LB000 ACC=LB001 DEC=LB001
MOVL C00202 V=17 PL=LB000 ACC=LB001 DEC=LB001
MOVL C00203 V=17 PL=LB000 ACC=LB001 DEC=LB001
MOVL C00204 V=17 PL=LB000 ACC=LB001 DEC=LB001
MOVL C00205 V=17 PL=LB000 ACC=LB001 DEC=LB001
MOVL C00206 V=17 PL=LB000 ACC=LB001 DEC=LB001
MOVL C00207 V=17 PL=LB000 ACC=LB001 DEC=LB001
MOVL C00208 V=17 PL=LB000 ACC=LB001 DEC=LB001
MOVL C00209 V=17 PL=LB000 ACC=LB001 DEC=LB001
MOVL C00210 V=17 PL=LB000 ACC=LB001 DEC=LB001
MOVL C00211 V=17 PL=LB000 ACC=LB001 DEC=LB001
MOVL C00212 V=17 PL=LB000 ACC=LB001 DEC=LB001
MOVL C00213 V=17 PL=LB000 ACC=LB001 DEC=LB001
MOVL C00214 V=17 PL=LB000 ACC=LB001 DEC=LB001
MOVL C00215 V=17 PL=LB000 ACC=LB001 DEC=LB001
MOVL C00216 V=17 PL=LB000 ACC=LB001 DEC=LB001
MOVL C00217 V=17 PL=LB000 ACC=LB001 DEC=LB001
MOVL C00218 V=17 PL=LB000 ACC=LB001 DEC=LB001
MOVL C00219 V=17 PL=LB000 ACC=LB001 DEC=LB001
MOVL C00220 V=17 PL=LB000 ACC=LB001 DEC=LB001
MOVL C00221 V=17 PL=LB000 ACC=LB001 DEC=LB001
MOVL C00222 V=17 PL=LB000 ACC=LB001 DEC=LB001
MOVL C00223 V=17 PL=LB000 ACC=LB001 DEC=LB001
MOVL C00224 V=17 PL=LB000 ACC=LB001 DEC=LB001
MOVL C00225 V=17 PL=LB000 ACC=LB001 DEC=LB001
MOVL C00226 V=17 PL=LB000 ACC=LB001 DEC=LB001
MOVL C00227 V=17 PL=LB000 ACC=LB001 DEC=LB001
MOVL C00228 V=17 PL=LB000 ACC=LB001 DEC=LB001
MOVL C00229 V=17 PL=LB000 ACC=LB001 DEC=LB001
MOVL C00230 V=17 PL=LB000 ACC=LB001 DEC=LB001
MOVL C00231 V=17 PL=LB000 ACC=LB001 DEC=LB001
MOVL C00232 V=17 PL=LB000 ACC=LB001 DEC=LB001
MOVL C00233 V=17 PL=LB000 ACC=LB001 DEC=LB001
MOVL C00234 V=17 PL=LB000 ACC=LB001 DEC=LB001
MOVL C00235 V=17 PL=LB000 ACC=LB001 DEC=LB001
MOVL C00236 V=17 PL=LB000 ACC=LB001 DEC=LB001
MOVL C00237 V=17 PL=LB000 ACC=LB001 DEC=LB001
MOVL C00238 V=17 PL=LB000 ACC=LB001 DEC=LB001
MOVL C00239 V=17 PL=LB000 ACC=LB001 DEC=LB001
MOVL C00240 V=17 PL=LB000 ACC=LB001 DEC=LB001
MOVL C00241 V=17 PL=LB000 ACC=LB001 DEC=LB001
MOVL C00242 V=17 PL=LB000 ACC=LB001 DEC=LB001
MOVL C00243 V=17 PL=LB000 ACC=LB001 DEC=LB001
MOVL C00244 V=17 PL=LB000 ACC=LB001 DEC=LB001
MOVL C00245 V=17 PL=LB000 ACC=LB001 DEC=LB001
MOVL C00246 V=17 PL=LB000 ACC=LB001 DEC=LB001
MOVL C00247 V=17 PL=LB000 ACC=LB001 DEC=LB001
MOVL C00248 V=17 PL=LB000 ACC=LB001 DEC=LB001
MOVL C00249 V=17 PL=LB000 ACC=LB001 DEC=LB001
MOVL C00250 V=17 PL=LB000 ACC=LB001 DEC=LB001
MOVL C00251 V=17 PL=LB000 ACC=LB001 DEC=LB001
MOVL C00252 V=17 PL=LB000 ACC=LB001 DEC=LB001
MOVL C00253 V=17 PL=LB000 ACC=LB001 DEC=LB001
MOVL C00254 V=17 PL=LB000 ACC=LB001 DEC=LB001
MOVL C00255 V=17 PL=LB000 ACC=LB001 DEC=LB001
MOVL C00256 V=17 PL=LB000 ACC=LB001 DEC=LB001
MOVL C00257 V=17 PL=LB000 ACC=LB001 DEC=LB001
MOVL C00258 V=17 PL=LB000 ACC=LB001 DEC=LB001
MOVL C00259 V=17 PL=LB000 ACC=LB001 DEC=LB001
MOVL C00260 V=17 PL=LB000 ACC=LB001 DEC=LB001
MOVL C00261 V=17 PL=LB000 ACC=LB001 DEC=LB001
MOVL C00262 V=17 PL=LB000 ACC=LB001 DEC=LB001
MOVL C00263 V=17 PL=LB000 ACC=LB001 DEC=LB001
MOVL C00264 V=17 PL=LB000 ACC=LB001 DEC=LB001
MOVL C00265 V=17 PL=LB000 ACC=LB001 DEC=LB001
MOVL C00266 V=17 PL=LB000 ACC=LB001 DEC=LB001
MOVL C00267 V=17 PL=LB000 ACC=LB001 DEC=LB001
MOVL C00268 V=17 PL=LB000 ACC=LB001 DEC=LB001
MOVL C00269 V=17 PL=LB000 ACC=LB001 DEC=LB001
MOVL C00270 V=17 PL=LB000 ACC=LB001 DEC=LB001
MOVL C00271 V=17 PL=LB000 ACC=LB001 DEC=LB001
MOVL C00272 V=17 PL=LB000 ACC=LB001 DEC=LB001
MOVL C00273 V=17 PL=LB000 ACC=LB001 DEC=LB001
MOVL C00274 V=17 PL=LB000 ACC=LB001 DEC=LB001
MOVL C00275 V=17 PL=LB000 ACC=LB001 DEC=LB001
MOVL C00276 V=17 PL=LB000 ACC=LB001 DEC=LB001
MOVL C00277 V=17 PL=LB000 ACC=LB001 DEC=LB001
MOVL C00278 V=17 PL=LB000 ACC=LB001 DEC=LB001
MOVL C00279 V=17 PL=LB000 ACC=LB001 DEC=LB001
MOVL C00280 V=17 PL=LB000 ACC=LB001 DEC=LB001
MOVL C00281 V=17 PL=LB000 ACC=LB001 DEC=LB001
MOVL C00282 V=17 PL=LB000 ACC=LB001 DEC=LB001
MOVL C00283 V=17 PL=LB000 ACC=LB001 DEC=LB001
MOVL C00284 V=17 PL=LB000 ACC=LB001 DEC=LB001
MOVL C00285 V=17 PL=LB000 ACC=LB001 DEC=LB001
MOVL C00286 V=17 PL=LB000 ACC=LB001 DEC=LB001
MOVL C00287 V=17 PL=LB000 ACC=LB001 DEC=LB001
MOVL C00288 V=17 PL=LB000 ACC=LB001 DEC=LB001
MOVL C00289 V=17 PL=LB000 ACC=LB001 DEC=LB001
MOVL C00290 V=17 PL=LB000 ACC=LB001 DEC=LB001
MOVL C00291 V=17 PL=LB000 ACC=LB001 DEC=LB001
MOVL C00292 V=17 PL=LB000 ACC=LB001 DEC=LB001
MOVL C00293 V=17 PL=LB000 ACC=LB001 DEC=LB001
MOVL C00294 V=17 PL=LB000 ACC=LB001 DEC=LB001
MOVL C00295 V=17 PL=LB000 ACC=LB001 DEC=LB001
MOVL C00296 V=17 PL=LB000 ACC=LB001 DEC=LB001
MOVL C00297 V=17 PL=LB000 ACC=LB001 DEC=LB001
MOVL C00298 V=17 PL=LB000 ACC=LB001 DEC=LB001
MOVL C00299 V=17 PL=LB000 ACC=LB001 DEC=LB001
MOVL C00300 V=17 PL=LB000 ACC=LB001 DEC=LB001
MOVL C00301 V=17 PL=LB000 ACC=LB001 DEC=LB001
MOVL C00302 V=17 PL=LB000 ACC=LB001 DEC=LB001
MOVL C00303 V=17 PL=LB000 ACC=LB001 DEC=LB001
MOVL C00304 V=17 PL=LB000 ACC=LB001 DEC=LB001
MOVL C00305 V=17 PL=LB000 ACC=LB001 DEC=LB001
MOVL C00306 V=17 PL=LB000 ACC=LB001 DEC=LB001
MOVL C00307 V=17 PL=LB000 ACC=LB001 DEC=LB001
MOVL C00308 V=17 PL=LB000 ACC=LB001 DEC=LB001
MOVL C00309 V=17 PL=LB000 ACC=LB001 DEC=LB001
MOVL C00310 V=17 PL=LB000 ACC=LB001 DEC=LB001
MOVL C00311 V=17 PL=LB000 ACC=LB001 DEC=LB001
MOVL C00312 V=17 PL=LB000 ACC=LB001 DEC=LB001
MOVL C00313 V=17 PL=LB000 ACC=LB001 DEC=LB001
MOVL C00314 V=17 PL=LB000 ACC=LB001 DEC=LB001
MOVL C00315 V=17 PL=LB000 ACC=LB001 DEC=LB001
MOVL C00316 V=17 PL=LB000 ACC=LB001 DEC=LB001
MOVL C00317 V=17 PL=LB000 ACC=LB001 DEC=LB001
MOVL C00318 V=17 PL=LB000 ACC=LB001 DEC=LB001
MOVL C00319 V=17 PL=LB000 ACC=LB001 DEC=LB001
MOVL C00320 V=17 PL=LB000 ACC=LB001 DEC=LB001
MOVL C00321 V=17 PL=LB000 ACC=LB001 DEC=LB001
MOVL C00322 V=17 PL=LB000 ACC=LB001 DEC=LB001
MOVL C00323 V=17 PL=LB000 ACC=LB001 DEC=LB001
MOVL C00324 V=17 PL=LB000 ACC=LB001 DEC=LB001
MOVL C00325 V=17 PL=LB000 ACC=LB001 DEC=LB001
MOVL C00326 V=17 PL=LB000 ACC=LB001 DEC=LB001
MOVL C00327 V=17 PL=LB000 ACC=LB001 DEC=LB001
MOVL C00328 V=17 PL=LB000 ACC=LB001 DEC=LB001
MOVL C00329 V=17 PL=LB000 ACC=LB001 DEC=LB001
MOVL C00330 V=17 PL=LB000 ACC=LB001 DEC=LB001
MOVL C00331 V=17 PL=LB000 ACC=LB001 DEC=LB001
MOVL C00332 V=17 PL=LB000 ACC=LB001 DEC=LB001
MOVL C00333 V=17 PL=LB000 ACC=LB001 DEC=LB001
MOVL C00334 V=17 PL=LB000 ACC=LB001 DEC=LB001
MOVL C00335 V=17 PL=LB000 ACC=LB001 DEC=LB001
MOVL C00336 V=17 PL=LB000 ACC=LB001 DEC=LB001
MOVL C00337 V=17 PL=LB000 ACC=LB001 DEC=LB001
MOVL C00338 V=17 PL=LB000 ACC=LB001 DEC=LB001
MOVL C00339 V=17 PL=LB000 ACC=LB001 DEC=LB001
MOVL C00340 V=17 PL=LB000 ACC=LB001 DEC=LB001
MOVL C00341 V=17 PL=LB000 ACC=LB001 DEC=LB001
MOVL C00342 V=17 PL=LB000 ACC=LB001 DEC=LB001
MOVL C00343 V=17 PL=LB000 ACC=LB001 DEC=LB001
MOVL C00344 V=17 PL=LB000 ACC=LB001 DEC=LB001
MOVL C00345 V=17 PL=LB000 ACC=LB001 DEC=LB001
MOVL C00346 V=17 PL=LB000 ACC=LB001 DEC=LB001
MOVL C00347 V=17 PL=LB000 ACC=LB001 DEC=LB001
MOVL C00348 V=17 PL=LB000 ACC=LB001 DEC=LB001
MOVL C00349 V=17 PL=LB000 ACC=LB001 DEC=LB001
MOVL C00350 V=17 PL=LB000 ACC=LB001 DEC=LB001
MOVL C00351 V=17 PL=LB000 ACC=LB001 DEC=LB001
MOVL C00352 V=17 PL=LB000 ACC=LB001 DEC=LB001
MOVL C00353 V=17 PL=LB000 ACC=LB001 DEC=LB001
MOVL C00354 V=17 PL=LB000 ACC=LB001 DEC=LB001
MOVL C00355 V=17 PL=LB000 ACC=LB001 DEC=LB001
MOVL C00356 V=17 PL=LB000 ACC=LB001 DEC=LB001
MOVL C00357 V=17 PL=LB000 ACC=LB001 DEC=LB001
MOVL C00358 V=17 PL=LB000 ACC=LB001 DEC=LB001
MOVL C00359 V=17 PL=LB000 ACC=LB001 DEC=LB001
MOVL C00360 V=17 PL=LB000 ACC=LB001 DEC=LB001
MOVL C00361 V=17 PL=LB000 ACC=LB001 DEC=LB001
MOVL C00362 V=17 PL=LB000 ACC=LB001 DEC=LB001
MOVL C00363 V=17 PL=LB000 ACC=LB001 DEC=LB001
MOVL C00364 V=17 PL=LB000 ACC=LB001 DEC=LB001
MOVL C00365 V=17 PL=LB000 ACC=LB001 DEC=LB001
MOVL C00366 V=17 PL=LB000 ACC=LB001 DEC=LB001
MOVL C00367 V=17 PL=LB000 ACC=LB001 DEC=LB001
MOVL C00368 V=17 PL=LB000 ACC=LB001 DEC=LB001
MOVL C00369 V=17 PL=LB000 ACC=LB001 DEC=LB001
MOVL C00370 V=17 PL=LB000 ACC=LB001 DEC=LB001
MOVL C00371 V=17 PL=LB000 ACC=LB001 DEC=LB001
MOVL C00372 V=17 PL=LB000 ACC=LB001 DEC=LB001
MOVL C00373 V=17 PL=LB000 ACC=LB001 DEC=LB001
MOVL C00374 V=17 PL=LB000 ACC=LB001 DEC=LB001
MOVL C00375 V=17 PL=LB000 ACC=LB001 DEC=LB001
MOVL C00376 V=17 PL=LB000 ACC=LB001 DEC=LB001
MOVL C00377 V=17 PL=LB000 ACC=LB001 DEC=LB001
MOVL C00378 V=17 PL=LB000 ACC=LB001 DEC=LB001
MOVL C00379 V=17 PL=LB000 ACC=LB001 DEC=LB001
MOVL C00380 V=17 PL=LB000 ACC=LB001 DEC=LB001
MOVL C00381 V=17 PL=LB000 ACC=LB001 DEC=LB001
MOVL C00382 V=17 PL=LB000 ACC=LB001 DEC=LB001
MOVL C00383 V=17 PL=LB000 ACC=LB001 DEC=LB001
MOVL C00384 V=17 PL=LB000 ACC=LB001 DEC=LB001
MOVL C00385 V=17 PL=LB000 ACC=LB001 DEC=LB001
MOVL C00386 V=17 PL=LB000 ACC=LB001 DEC=LB001
MOVL C00387 V=17 PL=LB000 ACC=LB001 DEC=LB001
MOVL C00388 V=17 PL=LB000 ACC=LB001 DEC=LB001
MOVL C00389 V=17 PL=LB000 ACC=LB001 DEC=LB001
MOVL C00390 V=17 PL=LB000 ACC=LB001 DEC=LB001
MOVL C00391 V=17 PL=LB000 ACC=LB001 DEC=LB001
MOVL C00392 V=17 PL=LB000 ACC=LB001 DEC=LB001
MOVL C00393 V=17 PL=LB000 ACC=LB001 DEC=LB001
MOVL C00394 V=17 PL=LB000 ACC=LB001 DEC=LB001
MOVL C00395 V=17 PL=LB000 ACC=LB001 DEC=LB001
MOVL C00396 V=17 PL=LB000 ACC=LB001 DEC=LB001
MOVL C00397 V=17 PL=LB000 ACC=LB001 DEC=LB001
MOVL C00398 V=17 PL=LB000 ACC=LB001 DEC=LB001
MOVL C00399 V=17 PL=LB000 ACC=LB001 DEC=LB001
MOVL C00400 V=17 PL=LB000 ACC=LB001 DEC=LB001
MOVL C00401 V=17 PL=LB000 ACC=LB001 DEC=LB001
MOVL C00402 V=17 PL=LB000 ACC=LB001 DEC=LB001
MOVL C00403 V=17 PL=LB000 ACC=LB001 DEC=LB001
MOVL C00404 V=17 PL=LB000 ACC=LB001 DEC=LB001
MOVL C00405 V=17 PL=LB000 ACC=LB001 DEC=LB001
MOVL C00406 V=17 PL=LB000 ACC=LB001 DEC=LB001
MOVL C00407 V=17 PL=LB000 ACC=LB001 DEC=LB001
MOVL C00408 V=17 PL=LB000 ACC=LB001 DEC=LB001
MOVL C00409 V=17 PL=LB000 ACC=LB001 DEC=LB001
MOVL C00410 V=17 PL=LB000 ACC=LB001 DEC=LB001
MOVL C00411 V=17 PL=LB000 ACC=LB001 DEC=LB001
MOVL C00412 V=17 PL=LB000 ACC=LB001 DEC=LB001
MOVL C00413 V=17 PL=LB000 ACC=LB001 DEC=LB001
MOVL C00414 V=17 PL=LB000 ACC=LB001 DEC=LB001
MOVL C00415 V=17 PL=LB000 ACC=LB001 DEC=LB001
MOVL C00416 V=17 PL=LB000 ACC=LB001 DEC=LB001
MOVL C00417 V=17 PL=LB000 ACC=LB001 DEC=LB001
MOVL C00418 V=17 PL=LB000 ACC=LB001 DEC=LB001
MOVL C00419 V=17 PL=LB000 ACC=LB001 DEC=LB001
MOVL C00420 V=17 PL=LB000 ACC=LB001 DEC=LB001
MOVL C00421 V=17 PL=LB000 ACC=LB001 DEC=LB001
MOVL C00422 V=17 PL=LB000 ACC=LB001 DEC=LB001
MOVL C00423 V=17 PL=LB000 ACC=LB001 DEC=LB001
MOVL C00424 V=17 PL=LB000 ACC=LB001 DEC=LB001
MOVL C00425 V=17 PL=LB000 ACC=LB001 DEC=LB001
MOVL C00426 V=17 PL=LB000 ACC=LB001 DEC=LB001
MOVL C00427 V=17 PL=LB000 ACC=LB001 DEC=LB001
MOVL C00428 V=17 PL=LB000 ACC=LB001 DEC=LB001
MOVL C00429 V=17 PL=LB000 ACC=LB001 DEC=LB001
MOVL C00430 V=17 PL=LB000 ACC=LB001 DEC=LB001
MOVL C00431 V=17 PL=LB000 ACC=LB001 DEC=LB001
MOVL C00432 V=17 PL=LB000 ACC=LB001 DEC=LB001
MOVL C00433 V=17 PL=LB000 ACC=LB001 DEC=LB001
MOVL C00434 V=17 PL=LB000 ACC=LB001 DEC=LB001
MOVL C00435 V=17 PL=LB000 ACC=LB001 DEC=LB001
MOVL C00436 V=17 PL=LB000 ACC=LB001 DEC=LB001
MOVL C00437 V=17 PL=LB000 ACC=LB001 DEC=LB001
MOVL C00438 V=17 PL=LB000 ACC=LB001 DEC=LB001
MOVL C00439 V=17 PL=LB000 ACC=LB001 DEC=LB001
MOVL C00440 V=17 PL=LB000 ACC=LB001 DEC=LB001
MOVL C00441 V=17 PL=LB000 ACC=LB001 DEC=LB001
MOVL C00442 V=17 PL=LB000 ACC=LB001 DEC=LB001
MOVL C00443 V=17 PL=LB000 ACC=LB001 DEC=LB001
MOVL C00444 V=17 PL=LB000 ACC=LB001 DEC=LB001
MOVL C00445 V=17 PL=LB000 ACC=LB001 DEC=LB001
MOVL C00446 V=17 PL=LB000 ACC=LB001 DEC=LB001
MOVL C00447 V=17 PL=LB000 ACC=LB001 DEC=LB001
MOVL C00448 V=17 PL=LB000 ACC=LB001 DEC=LB001
MOVL C00449 V=17 PL=LB000 ACC=LB001 DEC=LB001
MOVL C00450 V=17 PL=LB000 ACC=LB001 DEC=LB001
MOVL C00451 V=17 PL=LB000 ACC=LB001 DEC=LB001
MOVL C00452 V=17 PL=LB000 ACC=LB001 DEC=LB001
MOVL C00453 V=17 PL=LB000 ACC=LB001 DEC=LB001
MOVL C00454 V=17 PL=LB000 ACC=LB001 DEC=LB001
MOVL C00455 V=17 PL=LB000 ACC=LB001 DEC=LB001
MOVL C00456 V=17 PL=LB000 ACC=LB001 DEC=LB001
MOVL C00457 V=17 PL=LB000 ACC=LB001 DEC=LB001
MOVL C00458 V=17 PL=LB000 ACC=LB001 DEC=LB001
MOVL C00459 V=17 PL=LB000 ACC=LB001 DEC=LB001
MOVL C00460 V=17 PL=LB000 ACC=LB001 DEC=LB001
MOVL C00461 V=17 PL=LB000 ACC=LB001 DEC=LB001
MOVL C00462 V=17 PL=LB000 ACC=LB001 DEC=LB001
MOVL C00463 V=17 PL=LB000 ACC=LB001 DEC=LB001
MOVL C00464 V=17 PL=LB000 ACC=LB001 DEC=LB001
MOVL C00465 V=17 PL=LB000 ACC=LB001 DEC=LB001
MOVL C00466 V=17 PL=LB000 ACC=LB001 DEC=LB001
MOVL C00467 V=17 PL=LB000 ACC=LB001 DEC=LB001
MOVL C00468 V=17 PL=LB000 ACC=LB001 DEC=LB001
MOVL C00469 V=17 PL=LB000 ACC=LB001 DEC=LB001
MOVL C00470 V=17 PL=LB000 ACC=LB001 DEC=LB001
MOVL C00471 V=17 PL=LB000 ACC=LB001 DEC=LB001
MOVL C00472 V=17 PL=LB000 ACC=LB001 DEC=LB001
MOVL C00473 V=17 PL=LB000 ACC=LB001 DEC=LB001
MOVL C00474 V=17 PL=LB000 ACC=LB001 DEC=LB001
MOVL C00475 V=17 PL=LB000 ACC=LB001 DEC=LB001
MOVL C00476 V=17 PL=LB000 ACC=LB001 DEC=LB001
MOVL C00477 V=17 PL=LB000 ACC=LB001 DEC=LB001
MOVL C00478 V=17 PL=LB000 ACC=LB001 DEC=LB001
MOVL C00479 V=17 PL=LB000 ACC=LB001 DEC=LB001
' Lead Out Move Starts
MOVL C00480 V=17 PL=LB000 ACC=LB001 DEC=LB001
MOVL C00481 V=17 PL=LB000 ACC=LB001 DEC=LB001
MOVL C00482 V=17 PL=LB000 ACC=LB001 DEC=LB001
MOVL C00483 V=17 PL=LB000 ACC=LB001 DEC=LB001
MOVL C00484 V=17 PL=LB000 ACC=LB001 DEC=LB001
MOVL C00485 V=17 PL=LB000 ACC=LB001 DEC=LB001
MOVL C00486 V=17 PL=LB000 ACC=LB001 DEC=LB001
MOVL C00487 V=17 PL=LB000 ACC=LB001 DEC=LB001
MOVL C00488 V=17 PL=LB000 ACC=LB001 DEC=LB001
MOVL C00489 V=17 PL=LB000 ACC=LB001 DEC=LB001
MOVL C00490 V=17 PL=LB000 ACC=LB001 DEC=LB001
MOVL C00491 V=17 PL=LB000 ACC=LB001 DEC=LB001
MOVL C00492 V=17 PL=LB000 ACC=LB001 DEC=LB001
MOVL C00493 V=17 PL=LB000 ACC=LB001 DEC=LB001
MOVL C00494 V=17 PL=LB000 ACC=LB001 DEC=LB001
MOVL C00495 V=17 PL=LB000 ACC=LB001 DEC=LB001
MOVL C00496 V=17 PL=LB000 ACC=LB001 DEC=LB001
' Rapid Move Starts
MOVL C00497 V=17 PL=LB000 ACC=LB001 DEC=LB001
MOVL C00498 V=17 PL=LB000 ACC=LB001 DEC=LB001
' By Autodesk Fusion CAM 2.0.20494
' Tool = 8
' Spindle = 6000 RPM
' Set Position Level
' Set Acceleration
' Program Start
' First Toolpath Point
END
